# B&R Automation Studio project BenchEDM_AS6 (part 8)

#### OMD_MR.st
```iecst
ACTION OMD_MR:

	FOR i := 0 TO MAX_DRIVER_MR_IDX DO
		IF NOT gDriver.MR[i].FirstScanComplete THEN
			gDriver.MR[i].FirstScanComplete 			:= TRUE;
			gDriver.MR[i].DefaultPar.Device				:= 'SL2.IF1.ST1.IF1.ST5.IF1';					//ST
			gDriver.MR[i].DefaultPar.Mode				:= '/PHY=RS485 /PA=E /DB=8 /SB=1 /BD=38400';	//ST
			gDriver.MR[i].DefaultPar.DataObject			:= 'MbRTU';										//ST
			gDriver.MR[i].DefaultPar.IsAscii			:= FALSE;										//BO
			gDriver.MR[i].DefaultPar.Timeout			:= 1.0;											//LR
			gDriver.MR[i].DefaultPar.CmdNode			:= 1;											//UD
			gDriver.MR[i].DefaultPar.CmdFunctionCall	:= 1;											//UD
			gDriver.MR[i].DefaultPar.CmdOffset			:= 1;											//UD
			gDriver.MR[i].DefaultPar.CmdData			:= 0;											//UD
			brsmemcpy(ADR(gDriver.MR[i].Par),ADR(gDriver.MR[i].DefaultPar),SIZEOF(gDriver.MR[i].Par));
		ELSIF NOT gDriver.MR[i].ParametersLoaded AND gMain.Services.Recipes.Out.ParametersReady THEN
			gDriver.MR[i].ParametersLoaded := TRUE;
			brsmemcpy(ADR(gDriver.MR[i].Par),ADR(gPar.Driver.MR[i]),SIZEOF(gDriver.MR[i].Par));
		END_IF;

		brsmemset(ADR(gDriver.MR[i].Sev),0,SIZEOF(gDriver.MR[i].Sev));
		brsmemset(ADR(gDriver.MR[i].Status),0,SIZEOF(gDriver.MR[i].Status));
		FOR j := 0 TO MAX_DRIVER_MR_MON_IDX DO
			IF gDriver.MR[i].Par.Mon[j].Enable THEN
				IF gDriver.MR[i].Mon[j] THEN
					gDriver.MR[i].CTON_Mon[j](IN := TRUE, PT := LREAL_TO_TIME(gDriver.MR[i].Par.Mon[j].Time*1000.0));
					IF gDriver.MR[i].CTON_Mon[j].Q THEN
						gDriver.MR[i].Sev[j] := gDriver.MR[i].Par.Mon[j].Sev;
						IF gDriver.MR[i].Status.Severity < gDriver.MR[i].Sev[j] THEN
							gDriver.MR[i].Status.Severity := gDriver.MR[i].Sev[j];
						END_IF;
					END_IF;
				ELSE
					gDriver.MR[i].CTON_Mon[j](IN := FALSE);
					gDriver.MR[i].Sev[j] := 0;
				END_IF;
			ELSE
				gDriver.MR[i].CTON_Mon[j](IN := FALSE);
				gDriver.MR[i].Sev[j] := 0;
			END_IF;
		END_FOR;
		IF gDriver.MR[i].Cmd[C_MR_RESET] OR gDriver.ResetAll THEN
			gDriver.MR[i].Cmd[C_MR_RESET] := FALSE;
			brsmemset(ADR(gDriver.MR[i].Mon),0,SIZEOF(gDriver.MR[i].Mon));
			brsmemset(ADR(gDriver.MR[i].Cmd),0,SIZEOF(gDriver.MR[i].Cmd));
			brsmemset(ADR(gDriver.MR[i].Sev),0,SIZEOF(gDriver.MR[i].Sev));
			brsmemset(ADR(gDriver.MR[i].Status),0,SIZEOF(gDriver.MR[i].Status));
		END_IF;
		IF gDriver.MR[i].Cmd[C_MR_CLEARCMD] THEN
			gDriver.MR[i].Cmd[C_MR_CLEARCMD] := FALSE;
			brsmemset(ADR(gDriver.MR[i].Cmd),0,SIZEOF(gDriver.MR[i].Cmd));
		END_IF;
		IF gDriver.MR[i].Cmd[C_MR_CLEARMON] THEN
			gDriver.MR[i].Cmd[C_MR_CLEARMON] := FALSE;
			brsmemset(ADR(gDriver.MR[i].Status.Severity),0,SIZEOF(gDriver.MR[i].Status.Severity));
			brsmemset(ADR(gDriver.MR[i].Sev),0,SIZEOF(gDriver.MR[i].Sev));
			brsmemset(ADR(gDriver.MR[i].Par.Mon),0,SIZEOF(gDriver.MR[i].Par.Mon));
		END_IF;
		IF gDriver.MR[i].Cmd[C_MR_DEFAULTMON] THEN
			gDriver.MR[i].Cmd[C_MR_DEFAULTMON] := FALSE;
			brsmemcpy(ADR(gDriver.MR[i].Par.Mon),ADR(gDriver.MR[i].DefaultPar.Mon),SIZEOF(gDriver.MR[i].Par.Mon));
		END_IF;
		IF gDriver.MR[i].Cmd[C_MR_CLEARPAR] THEN
			gDriver.MR[i].Cmd[C_MR_CLEARPAR] := FALSE;
			brsmemset(ADR(gDriver.MR[i].Par),0,SIZEOF(gDriver.MR[i].Par));
		END_IF;
		IF gDriver.MR[i].Cmd[C_MR_DEFAULTPAR] THEN
			gDriver.MR[i].Cmd[C_MR_DEFAULTPAR] := FALSE;
			brsmemcpy(ADR(gDriver.MR[i].Par),ADR(gDriver.MR[i].DefaultPar),SIZEOF(gDriver.MR[i].Par));
		END_IF;
		IF gDriver.MR[i].Cmd[C_MR_SAVEPAR] THEN
			gDriver.MR[i].Cmd[C_MR_SAVEPAR] := FALSE;
			brsmemcpy(ADR(gPar.Driver.MR[i]),ADR(gDriver.MR[i].Par),SIZEOF(gDriver.MR[i].Par));
		END_IF;
		IF gDriver.MR[i].Cmd[C_MR_LOADPAR] THEN
			gDriver.MR[i].Cmd[C_MR_LOADPAR] := FALSE;
			brsmemcpy(ADR(gDriver.MR[i].Par),ADR(gPar.Driver.MR[i]),SIZEOF(gDriver.MR[i].Par));
		END_IF;

		gDriver.MR[i].MBMOpen_0.enable					:= gDriver.MR[i].Cmd[C_MR_MBMOPEN] AND NOT (gDriver.MR[i].Cmd[C_MR_ERRORRESET] OR gMain.ErrorReset);
		gDriver.MR[i].MBMaster_0.enable					:= gDriver.MR[i].Cmd[C_MR_MBMASTER] AND NOT (gDriver.MR[i].Cmd[C_MR_ERRORRESET] OR gMain.ErrorReset);
		gDriver.MR[i].MBMCmd_0.enable					:= gDriver.MR[i].Cmd[C_MR_MBMCMD] AND NOT (gDriver.MR[i].Cmd[C_MR_ERRORRESET] OR gMain.ErrorReset);
		gDriver.MR[i].MBMClose_0.enable					:= gDriver.MR[i].Cmd[C_MR_MBMCLOSE] AND NOT (gDriver.MR[i].Cmd[C_MR_ERRORRESET] OR gMain.ErrorReset);

		gDriver.MR[i].MBMOpen_0(pDevice := ADR(gDriver.MR[i].Par.Device), pMode := ADR(gDriver.MR[i].Par.Mode), pConfig := ADR(gDriver.MR[i].Par.DataObject), timeout := LREAL_TO_UINT(gDriver.MR[i].Par.Timeout*1000.0), ascii := BOOL_TO_USINT(gDriver.MR[i].Par.IsAscii));
		IF gDriver.MR[i].MBMOpen_0.ident <> 0 AND gDriver.MR[i].MBMOpen_0.enable THEN
			gDriver.MR[i].Ident := gDriver.MR[i].MBMOpen_0.ident;
		END_IF;
		gDriver.MR[i].MBMCmd_0(ident := gDriver.MR[i].Ident, mfc := UDINT_TO_USINT(gDriver.MR[i].Par.CmdFunctionCall), node := UDINT_TO_USINT(gDriver.MR[i].Par.CmdNode), data := ADR(gDriver.MR[i].Par.CmdData), offset := UDINT_TO_UINT(gDriver.MR[i].Par.CmdOffset), len := 1);
		gDriver.MR[i].MBMaster_0(ident := gDriver.MR[i].Ident);
		gDriver.MR[i].MBMClose_0(ident := gDriver.MR[i].Ident);
		IF gDriver.MR[i].MBMClose_0.enable AND gDriver.MR[i].MBMClose_0.status = 0 THEN
			gDriver.MR[i].Ident := 0;
		END_IF;

		gDriver.MR[i].Status.Active						:= gDriver.MR[i].MBMaster_0.enable AND (gDriver.MR[i].MBMaster_0.status = 65535 OR gDriver.MR[i].MBMaster_0.status = 0);

		gDriver.MR[i].Wait[W_MR_NOERROR]				:= BOOL_TO_DINT((gDriver.MR[i].MBMOpen_0.status = 0 OR gDriver.MR[i].MBMOpen_0.status = 65535 OR gDriver.MR[i].MBMOpen_0.status = 65534) AND (gDriver.MR[i].MBMaster_0.status = 0 OR gDriver.MR[i].MBMaster_0.status = 65535 OR gDriver.MR[i].MBMaster_0.status = 65534) AND (gDriver.MR[i].MBMCmd_0.status = 0 OR gDriver.MR[i].MBMCmd_0.status = 65535 OR gDriver.MR[i].MBMCmd_0.status = 65534) AND (gDriver.MR[i].MBMClose_0.status = 0 OR gDriver.MR[i].MBMClose_0.status = 65535 OR gDriver.MR[i].MBMClose_0.status = 65534));
		gDriver.MR[i].Wait[W_MR_MBMOPEN]				:= BOOL_TO_DINT(gDriver.MR[i].MBMOpen_0.status = 0);
		gDriver.MR[i].Wait[W_MR_MBMASTER]				:= BOOL_TO_DINT(gDriver.MR[i].MBMaster_0.status = 0 OR gDriver.MR[i].MBMaster_0.status = 65535);
		gDriver.MR[i].Wait[W_MR_MBMCMD]					:= BOOL_TO_DINT(gDriver.MR[i].MBMCmd_0.status = 0);
		gDriver.MR[i].Wait[W_MR_MBMCLOSE]				:= BOOL_TO_DINT(gDriver.MR[i].MBMClose_0.status = 0);

		IF gDriver.MR[i].MBMaster_0.enable THEN
			IF gDriver.MR[i].Wait[W_MR_NOERROR] = 0 THEN
				gDriver.MR[i].Mon[M_MR_ERROR]			:= TRUE;
			ELSIF gDriver.MR[i].MBMaster_0.execute THEN
				gDriver.MR[i].Mon[M_MR_ERROR]			:= FALSE;
			END_IF;
		ELSE
			gDriver.MR[i].Mon[M_MR_ERROR]				:= gDriver.MR[i].Wait[W_MR_NOERROR] = 0;
		END_IF;
	END_FOR;

END_ACTION
```

#### OMD_BX.st
```iecst
ACTION OMD_BX:

	FOR i := 0 TO MAX_DRIVER_BX_IDX DO
		IF NOT gDriver.BX[i].FirstScanComplete THEN
			gDriver.BX[i].FirstScanComplete 				:= TRUE;
			gDriver.BX[i].DefaultPar.EdgeFindMode			:= FALSE; 	//BO
			gDriver.BX[i].DefaultPar.ISOPulseMode			:= FALSE; 	//BO
			gDriver.BX[i].DefaultPar.ElectrodePositiveMode	:= FALSE; 	//BO
			gDriver.BX[i].DefaultPar.Current				:= 15.0; 	//RR
			gDriver.BX[i].DefaultPar.OnTime					:= 3.0; 	//RR
			gDriver.BX[i].DefaultPar.OffTime				:= 27.0; 	//RR
			gDriver.BX[i].DefaultPar.SetFeedback			:= 75.0; 	//RR
			gDriver.BX[i].DefaultPar.MinOverrideFactor		:= -200.0; 	//RR
			gDriver.BX[i].DefaultPar.MaxOverrideFactor		:= 200.0; 	//RR
			gDriver.BX[i].DefaultPar.PID.Gain				:= 0.1; 	//RR
			gDriver.BX[i].DefaultPar.PID.IntegrationTime	:= 0.0; 	//RR
			gDriver.BX[i].DefaultPar.PID.DerivativeTime		:= 0.0; 	//RR
			gDriver.BX[i].DefaultPar.PID.FilterTime			:= 0.0; 	//RR
			brsmemcpy(ADR(gDriver.BX[i].Par),ADR(gDriver.BX[i].DefaultPar),SIZEOF(gDriver.BX[i].Par));
		ELSIF NOT gDriver.BX[i].ParametersLoaded AND gMain.Services.Recipes.Out.ParametersReady THEN
			gDriver.BX[i].ParametersLoaded 					:= TRUE;
			brsmemcpy(ADR(gDriver.BX[i].Par),ADR(gPar.Driver.BX[i]),SIZEOF(gDriver.BX[i].Par));
		END_IF;

		brsmemset(ADR(gDriver.BX[i].Sev),0,SIZEOF(gDriver.BX[i].Sev));
		brsmemset(ADR(gDriver.BX[i].Status),0,SIZEOF(gDriver.BX[i].Status));
		FOR j := 0 TO MAX_DRIVER_BX_MON_IDX DO
			IF gDriver.BX[i].Par.Mon[j].Enable THEN
				IF gDriver.BX[i].Mon[j] THEN
					gDriver.BX[i].CTON_Mon[j](IN := TRUE, PT := LREAL_TO_TIME(gDriver.BX[i].Par.Mon[j].Time*1000.0));
					IF gDriver.BX[i].CTON_Mon[j].Q THEN
						gDriver.BX[i].Sev[j] 				:= gDriver.BX[i].Par.Mon[j].Sev;
						IF gDriver.BX[i].Status.Severity < gDriver.BX[i].Sev[j] THEN
							gDriver.BX[i].Status.Severity 	:= gDriver.BX[i].Sev[j];
						END_IF;
					END_IF;
				ELSE
					gDriver.BX[i].CTON_Mon[j](IN := FALSE);
					gDriver.BX[i].Sev[j] 					:= 0;
				END_IF;
			ELSE
				gDriver.BX[i].CTON_Mon[j](IN := FALSE);
				gDriver.BX[i].Sev[j] 						:= 0;
			END_IF;
		END_FOR;
		IF gDriver.BX[i].Cmd[C_BX_RESET] OR gDriver.ResetAll THEN
			gDriver.BX[i].Cmd[C_BX_RESET] 					:= FALSE;
			brsmemset(ADR(gDriver.BX[i].Mon),0,SIZEOF(gDriver.BX[i].Mon));
			brsmemset(ADR(gDriver.BX[i].Cmd),0,SIZEOF(gDriver.BX[i].Cmd));
			brsmemset(ADR(gDriver.BX[i].Sev),0,SIZEOF(gDriver.BX[i].Sev));
			brsmemset(ADR(gDriver.BX[i].Status),0,SIZEOF(gDriver.BX[i].Status));
		END_IF;
		IF gDriver.BX[i].Cmd[C_BX_CLEARCMD] THEN
			gDriver.BX[i].Cmd[C_BX_CLEARCMD] 				:= FALSE;
			brsmemset(ADR(gDriver.BX[i].Cmd),0,SIZEOF(gDriver.BX[i].Cmd));
		END_IF;
		IF gDriver.BX[i].Cmd[C_BX_CLEARMON] THEN
			gDriver.BX[i].Cmd[C_BX_CLEARMON] 				:= FALSE;
			brsmemset(ADR(gDriver.BX[i].Status.Severity),0,SIZEOF(gDriver.BX[i].Status.Severity));
			brsmemset(ADR(gDriver.BX[i].Sev),0,SIZEOF(gDriver.BX[i].Sev));
			brsmemset(ADR(gDriver.BX[i].Par.Mon),0,SIZEOF(gDriver.BX[i].Par.Mon));
		END_IF;
		IF gDriver.BX[i].Cmd[C_BX_DEFAULTMON] THEN
			gDriver.BX[i].Cmd[C_BX_DEFAULTMON] 				:= FALSE;
			brsmemcpy(ADR(gDriver.BX[i].Par.Mon),ADR(gDriver.BX[i].DefaultPar.Mon),SIZEOF(gDriver.BX[i].Par.Mon));
		END_IF;
		IF gDriver.BX[i].Cmd[C_BX_CLEARPAR] THEN
			gDriver.BX[i].Cmd[C_BX_CLEARPAR] 				:= FALSE;
			brsmemset(ADR(gDriver.BX[i].Par),0,SIZEOF(gDriver.BX[i].Par));
		END_IF;
		IF gDriver.BX[i].Cmd[C_BX_DEFAULTPAR] THEN
			gDriver.BX[i].Cmd[C_BX_DEFAULTPAR] 				:= FALSE;
			brsmemcpy(ADR(gDriver.BX[i].Par),ADR(gDriver.BX[i].DefaultPar),SIZEOF(gDriver.BX[i].Par));
		END_IF;
		IF gDriver.BX[i].Cmd[C_BX_SAVEPAR] THEN
			gDriver.BX[i].Cmd[C_BX_SAVEPAR] 				:= FALSE;
			brsmemcpy(ADR(gPar.Driver.BX[i]),ADR(gDriver.BX[i].Par),SIZEOF(gDriver.BX[i].Par));
		END_IF;
		IF gDriver.BX[i].Cmd[C_BX_LOADPAR] THEN
			gDriver.BX[i].Cmd[C_BX_LOADPAR] 				:= FALSE;
			brsmemcpy(ADR(gDriver.BX[i].Par),ADR(gPar.Driver.BX[i]),SIZEOF(gDriver.BX[i].Par));
		END_IF;

		gDriver.BX[i].Status.SetOffTime						:= gDriver.BX[i].Par.OffTime;
		gDriver.BX[i].Status.SetOnTime						:= gDriver.BX[i].Par.OnTime;
		gDriver.BX[i].Status.SetCurrent						:= gDriver.BX[i].Par.Current;
		gDriver.BX[i].Status.SetFeedback					:= gDriver.BX[i].Par.SetFeedback;
		gDriver.BX[i].Status.ActualPower					:= LREAL_TO_REAL(gIO.BX18.TC_IO_AI_Power.Signal.Filtered);
		gDriver.BX[i].Status.ActualFeedback					:= LREAL_TO_REAL(gIO.BX18.TC_IO_AI_Feedback.Signal.Filtered);
		gDriver.BX[i].Status.OutputActive					:= gIO.BX18.TC_IO_DI_EDMOutputActive.Signal.Filtered;
		gDriver.BX[i].Status.EdgeFindEnabled				:= gIO.BX18.TC_IO_DI_EdgefindModeEnabled.Signal.Filtered;
		gDriver.BX[i].Status.EdgeFound						:= gIO.BX18.TC_IO_DI_EdgeFound.Signal.Filtered;
		gDriver.BX[i].Status.StateInvalid					:= gIO.BX18.TC_IO_DI_ReqStateInvalid.Signal.Filtered;
		gDriver.BX[i].Status.SettingsInvalid				:= gIO.BX18.TC_IO_DI_ReqSettingsInvalid.Signal.Filtered;
		gDriver.BX[i].Status.PowerFault						:= gIO.BX18.TC_IO_DI_PowerFault.Signal.Filtered;
		gDriver.BX[i].Status.LowVoltageFault				:= gIO.BX18.TC_IO_DI_LowVoltageFault.Signal.Filtered;
		gDriver.BX[i].Status.HighVoltageFault				:= gIO.BX18.TC_IO_DI_HighVoltageFault.Signal.Filtered;
		gDriver.BX[i].Status.EstopActive					:= gIO.BX18.TC_IO_DI_EstopActive.Signal.Filtered;
		gDriver.BX[i].Status.ISOPulseMode					:= gIO.BX18.TC_IO_DI_ISOPulseMode.Signal.Filtered;
		gDriver.BX[i].Status.ElectrodePositiveMode			:= gIO.BX18.TC_IO_DI_ElectrodePositiveMode.Signal.Filtered;

		IF gDriver.BX[i].MTBasicsPID_0.PIDParameters.Gain <> gDriver.BX[i].Par.PID.Gain OR gDriver.BX[i].MTBasicsPID_0.PIDParameters.IntegrationTime <> gDriver.BX[i].Par.PID.IntegrationTime OR gDriver.BX[i].MTBasicsPID_0.PIDParameters.DerivativeTime <> gDriver.BX[i].Par.PID.DerivativeTime OR gDriver.BX[i].MTBasicsPID_0.PIDParameters.FilterTime <> gDriver.BX[i].Par.PID.FilterTime OR gDriver.BX[i].MTBasicsPID_0.MinOut <> gDriver.BX[i].Par.MinOverrideFactor OR gDriver.BX[i].MTBasicsPID_0.MaxOut <> gDriver.BX[i].Par.MaxOverrideFactor THEN
			gDriver.BX[i].MTBasicsPID_0.Update 				:= TRUE;
		END_IF;
		gDriver.BX[i].MTBasicsPID_0(Enable := gDriver.BX[i].Cmd[C_BX_ENABLE] AND gDriver.BX[i].Wait[W_BX_NOERROR] = 1, PIDParameters := gDriver.BX[i].Par.PID, MinOut := gDriver.BX[i].Par.MinOverrideFactor, MaxOut := gDriver.BX[i].Par.MaxOverrideFactor, SetValue := gDriver.BX[i].Par.SetFeedback, ActValue := gDriver.BX[i].Status.ActualFeedback, Invert := TRUE);
		gDriver.BX[i].MTBasicsPID_0.Update 					:= FALSE;

		gDriver.BX[i].Status.OverrideFactor					:= gDriver.BX[i].MTBasicsPID_0.Out;

		gDriver.BX[i].Wait[W_BX_NOERROR]					:= BOOL_TO_DINT(NOT gDriver.BX[i].Status.StateInvalid AND NOT gDriver.BX[i].Status.SettingsInvalid AND NOT gDriver.BX[i].Status.PowerFault AND NOT gDriver.BX[i].Status.LowVoltageFault AND NOT gDriver.BX[i].Status.HighVoltageFault AND NOT gDriver.BX[i].Status.EstopActive);
		gDriver.BX[i].Wait[W_BX_ACTIVE]						:= BOOL_TO_DINT(gDriver.BX[i].Wait[W_BX_NOERROR] = 1 AND gDriver.BX[i].Status.OutputActive);
		gDriver.BX[i].Mon[M_BX_ERROR]						:= gDriver.BX[i].Wait[W_BX_NOERROR] <> 1;

		gIO.BX18.TC_IO_AO_Current.Logical					:= gDriver.BX[i].Par.Current;
		gIO.BX18.TC_IO_AO_OffTime.Logical					:= gDriver.BX[i].Par.OffTime;
		gIO.BX18.TC_IO_AO_OnTime.Logical					:= gDriver.BX[i].Par.OnTime;
		gIO.BX18.TC_IO_DO_ChangeRequest.Logical				:= gIO.BX18.TC_IO_DI_CurrentChanged.Signal.Filtered OR gIO.BX18.TC_IO_DI_OnTimeChanged.Signal.Filtered OR gIO.BX18.TC_IO_DI_OffTimeChanged.Signal.Filtered;
		gIO.BX18.TC_IO_DO_EdgeFindMode.Logical				:= gDriver.BX[i].Par.EdgeFindMode;
		gIO.BX18.TC_IO_DO_ElectrodePositiveMode.Logical		:= gDriver.BX[i].Par.ElectrodePositiveMode;
		gIO.BX18.TC_IO_DO_ISOFreqMode.Logical				:= gDriver.BX[i].Par.ISOPulseMode;
		gIO.BX18.TC_IO_DO_Enable.Logical					:= gDriver.BX[i].Cmd[C_BX_ENABLE];
	END_FOR;

END_ACTION
```

#### OMD_IO.st - not listed in the package file held
```iecst
ACTION OMD_IO:

	FOR i := 0 TO MAX_DRIVER_AB_IDX DO
		IF NOT gDriver.AB[i].FirstScanComplete THEN
			gDriver.AB[i].FirstScanComplete 													:= TRUE;
			gDriver.AB[i].DefaultPar.AB.Acceleration											:= 50.0;							//RR
			gDriver.AB[i].DefaultPar.AB.AutoTune.FeedForward.Acceleration						:= 50.0;							//RR
			gDriver.AB[i].DefaultPar.AB.AutoTune.FeedForward.Direction							:= mcDIR_BOTH;						//McDirectionEnum
			gDriver.AB[i].DefaultPar.AB.AutoTune.FeedForward.MaxVelocityPercent					:= 50.0;							//RR
			gDriver.AB[i].DefaultPar.AB.AutoTune.FeedForward.Mode								:= mcACPAX_TUNE_FF_MODE_STANDARD; 	//McAcpAxAutoTuneFeedFwdModeEnum
			gDriver.AB[i].DefaultPar.AB.AutoTune.LoopFilterMode									:= mcAXIS_TUNE_LOOP_FILTER_F1;		//MpAxisAutoTuneLoopFilterModeEnum
			gDriver.AB[i].DefaultPar.AB.AutoTune.MaxCurrentPercent								:= 80.0;							//RR
			gDriver.AB[i].DefaultPar.AB.AutoTune.MaxDistance									:= 0.0;								//LR
			gDriver.AB[i].DefaultPar.AB.AutoTune.MaxPositionError								:= 1.0;								//LR
			gDriver.AB[i].DefaultPar.AB.AutoTune.Mode											:= mcAXIS_TUNE_AUTOMATIC;			//MpAxisAutoTuneModeEnum
			gDriver.AB[i].DefaultPar.AB.AutoTune.Options.MaxProportionalGain					:= 0.0;								//RR
			gDriver.AB[i].DefaultPar.AB.AutoTune.Options.SpeedTuneFilterTmeMode					:= mcACPAX_FILTER_TIME_USE;			//McAcpAxFilterTimeModeEnum
			gDriver.AB[i].DefaultPar.AB.AutoTune.Options.SpeedTuneLoopFilter1Mode				:= mcACPAX_LOOP_FILTER_IGNORE;		//McAcpAxLoopFilterModeEnum
			gDriver.AB[i].DefaultPar.AB.AutoTune.Orientation									:= mcACPAX_ORIENTATION_HORIZONTAL;	//McAcpAxAutoTuneOrientationEnum
			gDriver.AB[i].DefaultPar.AB.AutoTune.SaveControllerSettings							:= FALSE;							//BO
			gDriver.AB[i].DefaultPar.AB.Deceleration											:= 50.0;							//RR
			gDriver.AB[i].DefaultPar.AB.Direction												:= mcDIR_SHORTEST_WAY;				//McDirectionEnum
			gDriver.AB[i].DefaultPar.AB.Distance												:= 0.0;								//LR
			gDriver.AB[i].DefaultPar.AB.Homing.Mode												:= mcHOMING_DIRECT;					//McHomingModeEnum
			gDriver.AB[i].DefaultPar.AB.Homing.Position											:= 0.0;								//RR
			gDriver.AB[i].DefaultPar.AB.Homing.Options.Acceleration								:= 50.0;							//RR
			gDriver.AB[i].DefaultPar.AB.Homing.Options.AdditionalTorqueLimit.NegativeDirection	:= 0.0;								//RR
			gDriver.AB[i].DefaultPar.AB.Homing.Options.AdditionalTorqueLimit.PositiveDirection	:= 0.0;								//RR
			gDriver.AB[i].DefaultPar.AB.Homing.Options.BlockDetectionPositionError				:= 0.0;								//RR
			gDriver.AB[i].DefaultPar.AB.Homing.Options.DisableRestorePositionOnEnable			:= mcSWITCH_OFF;					//McSwitchEnum
			gDriver.AB[i].DefaultPar.AB.Homing.Options.DriveSpecificHoming						:= mcSWITCH_OFF;					//McSwitchEnum
			gDriver.AB[i].DefaultPar.AB.Homing.Options.DriveSpecificHomingMode					:= 0;								//SS
			gDriver.AB[i].DefaultPar.AB.Homing.Options.HomingDirection							:= mcDIR_POSITIVE;					//McDirectionEnum
			gDriver.AB[i].DefaultPar.AB.Homing.Options.HomingVelocity							:= 5.0;								//RR
			gDriver.AB[i].DefaultPar.AB.Homing.Options.KeepDirection							:= mcSWITCH_OFF;					//McSwitchEnum
			gDriver.AB[i].DefaultPar.AB.Homing.Options.PositionErrorStopLimit					:= 0.0;								//RR
			gDriver.AB[i].DefaultPar.AB.Homing.Options.ReferencePulse							:= mcSWITCH_OFF;					//McSwitchEnum
			gDriver.AB[i].DefaultPar.AB.Homing.Options.ReferencePulseBlockingDistance			:= 0.0;								//RR
			gDriver.AB[i].DefaultPar.AB.Homing.Options.RestorePositionVariableAddress			:= 0;								//UD
			gDriver.AB[i].DefaultPar.AB.Homing.Options.SensorOffset								:= 0.0;								//LR
			gDriver.AB[i].DefaultPar.AB.Homing.Options.SensorOffsetDirection					:= mcDIR_POSITIVE;					//McDirectionEnum
			gDriver.AB[i].DefaultPar.AB.Homing.Options.StartDirection							:= mcDIR_POSITIVE;					//McDirectionEnum
			gDriver.AB[i].DefaultPar.AB.Homing.Options.StartVelocity							:= 1.0;								//RR
			gDriver.AB[i].DefaultPar.AB.Homing.Options.SwitchEdge								:= mcDIR_POSITIVE;					//McDirectionEnum
			gDriver.AB[i].DefaultPar.AB.Homing.Options.TorqueLimit								:= 0.1;								//RR
			gDriver.AB[i].DefaultPar.AB.Jerk													:= 0.0;								//RR
			gDriver.AB[i].DefaultPar.AB.Jog.Acceleration										:= 50.0;							//RR
			gDriver.AB[i].DefaultPar.AB.Jog.Deceleration										:= 50.0;							//RR
			gDriver.AB[i].DefaultPar.AB.Jog.Jerk												:= 0.0;								//RR
			gDriver.AB[i].DefaultPar.AB.Jog.LimitPosition.FirstPosition							:= 0.0;								//LR
			gDriver.AB[i].DefaultPar.AB.Jog.LimitPosition.LastPosition							:= 0.0;								//LR
			gDriver.AB[i].DefaultPar.AB.Jog.Velocity											:= 5.0;								//RR
			gDriver.AB[i].DefaultPar.AB.LimitLoad.Direction										:= mcDIR_CURRENT;					//McDirectionEnum
			gDriver.AB[i].DefaultPar.AB.LimitLoad.Load											:= 2.0;								//RR
			gDriver.AB[i].DefaultPar.AB.Position												:= 0.0;								//LR
			gDriver.AB[i].DefaultPar.AB.Stop.Deceleration										:= 50.0;							//RR
			gDriver.AB[i].DefaultPar.AB.Stop.Jerk												:= 0.0;								//RR
			gDriver.AB[i].DefaultPar.AB.Stop.StopAtPosition.Activate							:= FALSE;							//BO
			gDriver.AB[i].DefaultPar.AB.Stop.StopAtPosition.Deceleration						:= 0.0;								//RR
			gDriver.AB[i].DefaultPar.AB.Stop.StopAtPosition.Position							:= 0.0;								//LR
			gDriver.AB[i].DefaultPar.AB.Velocity												:= 5.0;								//RR

			brsmemcpy(ADR(gDriver.AB[i].Par),ADR(gDriver.AB[i].DefaultPar),SIZEOF(gDriver.AB[i].Par));
		END_IF;

		brsmemset(ADR(gDriver.AB[i].Sev),0,SIZEOF(gDriver.AB[i].Sev));
		brsmemset(ADR(gDriver.AB[i].Status),0,SIZEOF(gDriver.AB[i].Status));
		FOR j := 0 TO MAX_DRIVER_AB_MON_IDX DO
			IF gDriver.AB[i].Par.Mon[j].Enable THEN
				IF gDriver.AB[i].Mon[j] THEN
					gDriver.AB[i].CTON_Mon[j](IN := TRUE, PT := LREAL_TO_TIME(gDriver.AB[i].Par.Mon[j].Time*1000.0));
					IF gDriver.AB[i].CTON_Mon[j].Q THEN
						gDriver.AB[i].Sev[j] := gDriver.AB[i].Par.Mon[j].Sev;
						IF gDriver.AB[i].Status.Severity < gDriver.AB[i].Sev[j] THEN
							gDriver.AB[i].Status.Severity := gDriver.AB[i].Sev[j];
						END_IF;
					END_IF;
				ELSE
					gDriver.AB[i].CTON_Mon[j](IN := FALSE);
					gDriver.AB[i].Sev[j] := 0;
				END_IF;
			ELSE
				gDriver.AB[i].CTON_Mon[j](IN := FALSE);
				gDriver.AB[i].Sev[j] := 0;
			END_IF;
		END_FOR;
		IF gDriver.AB[i].Cmd[C_AB_RESET] THEN
			gDriver.AB[i].Cmd[C_AB_RESET] := FALSE;
			brsmemset(ADR(gDriver.AB[i].Cmd),0,SIZEOF(gDriver.AB[i].Cmd));
			brsmemset(ADR(gDriver.AB[i].Sev),0,SIZEOF(gDriver.AB[i].Sev));
			brsmemset(ADR(gDriver.AB[i].Status),0,SIZEOF(gDriver.AB[i].Status));
			brsmemcpy(ADR(gDriver.AB[i].Par),ADR(gDriver.AB[i].DefaultPar),SIZEOF(gDriver.AB[i].Par));
		END_IF;
		IF gDriver.AB[i].Cmd[C_AB_CLEARCMD] THEN
			gDriver.AB[i].Cmd[C_AB_CLEARCMD] := FALSE;
			brsmemset(ADR(gDriver.AB[i].Cmd),0,SIZEOF(gDriver.AB[i].Cmd));
		END_IF;
		IF gDriver.AB[i].Cmd[C_AB_CLEARMON] THEN
			gDriver.AB[i].Cmd[C_AB_CLEARMON] := FALSE;
			brsmemset(ADR(gDriver.AB[i].Status.Severity),0,SIZEOF(gDriver.AB[i].Status.Severity));
			brsmemset(ADR(gDriver.AB[i].Sev),0,SIZEOF(gDriver.AB[i].Sev));
			brsmemset(ADR(gDriver.AB[i].Par.Mon),0,SIZEOF(gDriver.AB[i].Par.Mon));
		END_IF;
		IF gDriver.AB[i].Cmd[C_AB_DEFAULTMON] THEN
			gDriver.AB[i].Cmd[C_AB_DEFAULTMON] := FALSE;
			brsmemcpy(ADR(gDriver.AB[i].Par.Mon),ADR(gDriver.AB[i].DefaultPar.Mon),SIZEOF(gDriver.AB[i].Par.Mon));
		END_IF;
		IF gDriver.AB[i].Cmd[C_AB_CLEARPAR] THEN
			gDriver.AB[i].Cmd[C_AB_CLEARPAR] := FALSE;
			brsmemset(ADR(gDriver.AB[i].Par),0,SIZEOF(gDriver.AB[i].Par));
		END_IF;
		IF gDriver.AB[i].Cmd[C_AB_DEFAULTPAR] THEN
			gDriver.AB[i].Cmd[C_AB_DEFAULTPAR] := FALSE;
			brsmemcpy(ADR(gDriver.AB[i].Par),ADR(gDriver.AB[i].DefaultPar),SIZEOF(gDriver.AB[i].Par));
		END_IF;
		gDriver.AB[i].MpAxisBasic_0.ErrorReset			:= gDriver.AB[i].Cmd[C_AB_ERRORRESET] OR gMain.ErrorReset;
		gDriver.AB[i].MpAxisBasic_0.Home				:= gDriver.AB[i].Cmd[C_AB_HOME];
		gDriver.AB[i].MpAxisBasic_0.Power				:= gDriver.AB[i].Cmd[C_AB_POWER];
		gDriver.AB[i].MpAxisBasic_0.Update				:= gDriver.AB[i].Cmd[C_AB_UPDATE];
		gDriver.AB[i].MpAxisBasic_0.AutoTune			:= gDriver.AB[i].Cmd[C_AB_AUTOTUNE];
		gDriver.AB[i].MpAxisBasic_0.JogPositive			:= gDriver.AB[i].Cmd[C_AB_JOGPOSITIVE];
		gDriver.AB[i].MpAxisBasic_0.JogNegative			:= gDriver.AB[i].Cmd[C_AB_JOGNEGATIVE];
		gDriver.AB[i].MpAxisBasic_0.LimitLoad			:= gDriver.AB[i].Cmd[C_AB_LIMITLOAD];
		gDriver.AB[i].MpAxisBasic_0.Stop				:= gDriver.AB[i].Cmd[C_AB_STOP];
		gDriver.AB[i].MpAxisBasic_0.MoveAbsolute		:= gDriver.AB[i].Cmd[C_AB_MOVEABSOLUTE];
		gDriver.AB[i].MpAxisBasic_0.MoveAdditive		:= gDriver.AB[i].Cmd[C_AB_MOVEADDITIVE];
		gDriver.AB[i].MpAxisBasic_0.MoveVelocity		:= gDriver.AB[i].Cmd[C_AB_MOVEVELOCITY];
		gDriver.AB[i].MpAxisBasic_0.ReleaseBrake		:= gDriver.AB[i].Cmd[C_AB_RELEASEBRAKE];
		gDriver.AB[i].MpAxisBasic_0.Simulate			:= gDriver.AB[i].Cmd[C_AB_SIMULATE];

		gDriver.AB[i].MpAxisBasic_0(MpLink := gDriver.AB[i].MpLinkADR, Enable := TRUE, Parameters := ADR(gDriver.AB[i].Par.AB));

		gDriver.AB[i].Status.Position					:= gDriver.AB[i].MpAxisBasic_0.Position;
		gDriver.AB[i].Status.Velocity					:= gDriver.AB[i].MpAxisBasic_0.Velocity;

		gDriver.AB[i].Wait[W_AB_NOERROR]				:= BOOL_TO_DINT(NOT gDriver.AB[i].MpAxisBasic_0.Error);
		gDriver.AB[i].Wait[W_AB_COMMUNICATIONREADY]		:= BOOL_TO_DINT(gDriver.AB[i].MpAxisBasic_0.Info.CommunicationReady);
		gDriver.AB[i].Wait[W_AB_READYTOPOWERON]			:= BOOL_TO_DINT(gDriver.AB[i].MpAxisBasic_0.Info.ReadyToPowerOn);
		gDriver.AB[i].Wait[W_AB_POWERON]				:= BOOL_TO_DINT(gDriver.AB[i].MpAxisBasic_0.PowerOn);
		gDriver.AB[i].Wait[W_AB_ISHOMED]				:= BOOL_TO_DINT(gDriver.AB[i].MpAxisBasic_0.IsHomed AND NOT gDriver.AB[i].MpAxisBasic_0.CommandBusy);
		gDriver.AB[i].Wait[W_AB_LIMITLOADACTIVE]		:= BOOL_TO_DINT(gDriver.AB[i].MpAxisBasic_0.LimitLoadReady);
		gDriver.AB[i].Wait[W_AB_MOVEDONE]				:= BOOL_TO_DINT(gDriver.AB[i].MpAxisBasic_0.MoveDone);
		gDriver.AB[i].Wait[W_AB_UPDATEDONE]				:= BOOL_TO_DINT(gDriver.AB[i].MpAxisBasic_0.UpdateDone);
		gDriver.AB[i].Wait[W_AB_AUTOTUNEDONE]			:= BOOL_TO_DINT(gDriver.AB[i].MpAxisBasic_0.AutoTuneDone);
		gDriver.AB[i].Wait[W_AB_BRAKERELEASED]			:= BOOL_TO_DINT(gDriver.AB[i].MpAxisBasic_0.BrakeReleased);
		gDriver.AB[i].Wait[W_AB_COMMANDABORTED]			:= BOOL_TO_DINT(gDriver.AB[i].MpAxisBasic_0.CommandAborted);
		gDriver.AB[i].Wait[W_AB_COMMANDBUSY]			:= BOOL_TO_DINT(gDriver.AB[i].MpAxisBasic_0.CommandBusy);
		gDriver.AB[i].Wait[W_AB_INPOSITION]				:= BOOL_TO_DINT(gDriver.AB[i].MpAxisBasic_0.InPosition);
		gDriver.AB[i].Wait[W_AB_INVELOCITY]				:= BOOL_TO_DINT(gDriver.AB[i].MpAxisBasic_0.InVelocity);
		gDriver.AB[i].Wait[W_AB_MOVEACTIVE]				:= BOOL_TO_DINT(gDriver.AB[i].MpAxisBasic_0.MoveActive);
		gDriver.AB[i].Wait[W_AB_STOPPED]				:= BOOL_TO_DINT(gDriver.AB[i].MpAxisBasic_0.Stopped);
		gDriver.AB[i].Wait[W_AB_JOGGING]				:= BOOL_TO_DINT(gDriver.AB[i].MpAxisBasic_0.Info.Jogging);
		gDriver.AB[i].Wait[W_AB_JOGLIMITREACHED]		:= BOOL_TO_DINT(gDriver.AB[i].MpAxisBasic_0.Info.JogLimitReached);
		gDriver.AB[i].Wait[W_AB_SIMULATION]				:= BOOL_TO_DINT(gDriver.AB[i].MpAxisBasic_0.Info.Simulation);

		gDriver.AB[i].Mon[M_AB_ERROR]					:= gDriver.AB[i].MpAxisBasic_0.Error;
		gDriver.AB[i].Mon[M_AB_NOTPOWERON]				:= NOT gDriver.AB[i].MpAxisBasic_0.PowerOn;
	END_FOR;

//	McDirectionEnum :
//	(
//		mcDIR_POSITIVE := 0,							(*Movement only in the positive direction *)
//		mcDIR_NEGATIVE := 1,							(*Movement only in the negative direction*)
//		mcDIR_CURRENT := 2,								(*Movement in the direction of the active movement*)
//		mcDIR_SHORTEST_WAY := 3,						(*Movement with the shortest distance to the target, either in positive or negative direction. The movement will be in the positive direction if the distance is the same in both directions*)
//		mcDIR_EXCEED_PERIOD := 8,						(*The end position can be located outside of the axis period. The axis period can be exited in the negative direction if the end position is also negative*)
//		mcDIR_UNDEFINED := 9,							(*Movement in undefined direction*)
//		mcDIR_BOTH := 10								(*Movement in both directions*)
//	);
//	McSwitchEnum :
//	(
//		mcSWITCH_OFF := 0,		 						(*State/Behavior selection switched off*)
//		mcSWITCH_ON := 1			 					(*State/Behavior selection switched on*)
//	);
//	McHomingModeEnum :
//	(
//		mcHOMING_DIRECT := 0,							(*Direct homing. "Position" is used directly as the new axis position*)
//		mcHOMING_SWITCH_GATE := 1,						(*Homing with reference gate*)
//		mcHOMING_ABSOLUTE_SWITCH := 2,					(*Performs homing with absolute reference switch*)
//		mcHOMING_LIMIT_SWITCH := 4,	    				(*Homing with hardware limit switch*)
//		mcHOMING_ABSOLUTE := 5,							(*Homing by setting the "Position" homing offset for an absolute encoder*)
//		mcHOMING_DCM := 7,								(*Homing using interval-encoded reference marks*)
//		mcHOMING_BLOCK_TORQUE := 9,						(*Performs homing to mechanical limit, torque as criteria*)
//		mcHOMING_BLOCK_LAG_ERROR := 10,					(*Performs homing to mechanical limit, lag error as criteria*)
//		mcHOMING_ABSOLUTE_CORRECTION := 133,  			(*Homing by setting the "Position" homing offset for an absolute encoder with counter range correction. This mode must be used if the overflow of the absolute encoder is within the axis range of movement*)
//		mcHOMING_DCM_CORRECTION := 135,	 				(*Homing using distance-coded reference marks with counting range correction*)
//		mcHOMING_DEFAULT := 140,		 				(*All parameters, including "Position", are taken from the initial configuration for the axis*)
//		mcHOMING_INIT := 141,							(*All parameters, including "Position", are taken from an earlier initialization made using function block MC_BR_InitHome*)
//		mcHOMING_RESTORE_POSITION := 142				(*Restores position from a remanent variable*)
//	);
//	MpAxisAutoTuneModeEnum :
//	(
//		mcAXIS_TUNE_AUTOMATIC := 0, 					(* Performs a complete auto-tuning sequence of all controllers*)
//		mcAXIS_TUNE_SPEED := 1, 						(* Speed controller tuning*)
//		mcAXIS_TUNE_POSITION := 2, 						(* Position controller tuning*)
//		mcAXIS_TUNE_TEST := 3, 							(* Tests system stability*)
//		mcAXIS_TUNE_LOOP_FILTER := 4, 					(* Loop filter tuning*)
//		mcAXIS_TUNE_FEED_FORWARD := 5 					(*Feed forward tuning*)
//	);
//	MpAxisAutoTuneLoopFilterModeEnum :
//	(
//		mcAXIS_TUNE_LOOP_FILTER_F1 := 0, 				(*Tuning of loop filter 1 as a notch filter*)
//		mcAXIS_TUNE_LOOP_FILTER_F1_F2 := 1, 			(*Tuning of filter 1 and 2 as a notch filter*)
//		mcAXIS_TUNE_LOOP_FILTER_F1_F2_F3 := 2 			(*Tuning of filter 1, 2 and 3 as a notch filter*)
//	);
//	McAcpAxAutoTuneOrientationEnum:
//	(
//		mcACPAX_ORIENTATION_HORIZONTAL := 0, 		 	(*Horizontal orientation*)
//		mcACPAX_ORIENTATION_VERTICAL := 1    		 	(*Vertical orientation*)
//	);
//	McAcpAxFilterTimeModeEnum:
//	(
//		mcACPAX_FILTER_TIME_USE := 0,  					(*The determination of filter time constants is disabled; however, filter time constants are taken into account for autotuning*)
//		mcACPAX_FILTER_TIME_TUNE_MODE1 := 1, 		 	(*The controlled variable is the unfiltered actual speed n*)
//		mcACPAX_FILTER_TIME_TUNE_MODE2 := 2  		 	(*The controlled variable is the filtered actual speed n*)
//	);
//	McAcpAxLoopFilterModeEnum:
//	(
//		mcACPAX_LOOP_FILTER_IGNORE := 0,  				(*Loop filters are neither taken into account nor calculated.*)
//		mcACPAX_LOOP_FILTER_USE := 1,  					(*The parameters for all loop filters are taken into account for autotuning*)
//		mcACPAX_LOOP_FILTER_TUNE_NOTCH := 2  			(*The parameters for the loop filter are calculated*)
//	);
//	McAcpAxAutoTuneFeedFwdModeEnum:
//	(
//		mcACPAX_TUNE_FF_MODE_STANDARD := 0, 			(*Standard (active) tuning mode*)
//		mcACPAX_TUNE_FF_MODE_PASSIVE := 1 				(*Passive tuning mode*)
//	);
//	McAcpAxAutoTuneFeedFwdCmdEnum:
//	(
//		mcACPAX_TUNE_FF_CMD_START := 0, 				(*Start (standard or passive) tuning process*)
//		mcACPAX_TUNE_FF_CMD_FINISH := 1, 				(*Finish (passive) tuning process*)
//		mcACPAX_TUNE_FF_CMD_ABORT := 2 					(*Abort (stop) (passive) tuning process*)
//	);

END_ACTION
```

### Program Logical/Services (IEC)

#### Main.st - Init, cyclic, exit code
```iecst
PROGRAM _INIT

	gMain.Services.DirMan.In.RefreshDelay										:= 10.0;

	gMain.Services.DirMan.In.DirDef[0].Valid									:= TRUE;
	gMain.Services.DirMan.In.DirDef[0].DirPath									:= '';
	gMain.Services.DirMan.In.DirDef[0].Sanitize.AllowUndefinedDir				:= FALSE;
	gMain.Services.DirMan.In.DirDef[0].Sanitize.SanitizeFilesByRoot				:= FALSE;
	gMain.Services.DirMan.In.DirDef[0].Sanitize.SanitizeFilesByExt				:= TRUE;
	gMain.Services.DirMan.In.DirDef[0].Sanitize.FileExtension					:= '.~';
	gMain.Services.DirMan.In.DirDef[0].Sanitize.FileRoot						:= '';
	gMain.Services.DirMan.In.DirDef[0].Sanitize.MaxFiles						:= 4294967295;
	gMain.Services.DirMan.In.DirDef[0].Sanitize.MaxSize							:= 4294967295;

	gMain.Services.DirMan.In.DirDef[1].Valid									:= TRUE;
	gMain.Services.DirMan.In.DirDef[1].DirPath									:= 'Machine';
	gMain.Services.DirMan.In.DirDef[1].Sanitize.AllowUndefinedDir				:= FALSE;
	gMain.Services.DirMan.In.DirDef[1].Sanitize.SanitizeFilesByRoot				:= FALSE;
	gMain.Services.DirMan.In.DirDef[1].Sanitize.SanitizeFilesByExt				:= TRUE;
	gMain.Services.DirMan.In.DirDef[1].Sanitize.FileExtension					:= '.txt';
	gMain.Services.DirMan.In.DirDef[1].Sanitize.FileRoot						:= '';
	gMain.Services.DirMan.In.DirDef[1].Sanitize.MaxFiles						:= 4294967295;
	gMain.Services.DirMan.In.DirDef[1].Sanitize.MaxSize							:= 4294967295;

	gMain.Services.DirMan.In.DirDef[2].Valid									:= TRUE;
	gMain.Services.DirMan.In.DirDef[2].DirPath									:= 'GCODE';
	gMain.Services.DirMan.In.DirDef[2].Sanitize.AllowUndefinedDir				:= FALSE;
	gMain.Services.DirMan.In.DirDef[2].Sanitize.SanitizeFilesByRoot				:= FALSE;
	gMain.Services.DirMan.In.DirDef[2].Sanitize.SanitizeFilesByExt				:= FALSE;
	gMain.Services.DirMan.In.DirDef[2].Sanitize.FileExtension					:= '';
	gMain.Services.DirMan.In.DirDef[2].Sanitize.FileRoot						:= '';
	gMain.Services.DirMan.In.DirDef[2].Sanitize.MaxFiles						:= 100;
	gMain.Services.DirMan.In.DirDef[2].Sanitize.MaxSize							:= 4294967295;

	gMain.Services.DirMan.In.DirDef[3].Valid									:= TRUE;
	gMain.Services.DirMan.In.DirDef[3].DirPath									:= 'AlarmHistory';
	gMain.Services.DirMan.In.DirDef[3].Sanitize.AllowUndefinedDir				:= FALSE;
	gMain.Services.DirMan.In.DirDef[3].Sanitize.SanitizeFilesByRoot				:= TRUE;
	gMain.Services.DirMan.In.DirDef[3].Sanitize.SanitizeFilesByExt				:= TRUE;
	gMain.Services.DirMan.In.DirDef[3].Sanitize.FileExtension					:= '.csv';
	gMain.Services.DirMan.In.DirDef[3].Sanitize.FileRoot						:= 'Alarms';
	gMain.Services.DirMan.In.DirDef[3].Sanitize.MaxFiles						:= 10;
	gMain.Services.DirMan.In.DirDef[3].Sanitize.MaxSize							:= 4294967295;

	gMain.Services.Recipes.In.RecipeDefinitions[0].MpLink						:= gRecipeXml_Rem;
	gMain.Services.Recipes.In.RecipeDefinitions[0].DeviceName					:= gMain.Services.DeviceName;
	gMain.Services.Recipes.In.RecipeDefinitions[0].FileName						:= 'Machine/gRem.txt';
	gMain.Services.Recipes.In.RecipeDefinitions[0].VarName						:= 'gRem';
	gMain.Services.Recipes.In.RecipeDefinitions[0].pVar							:= ADR(gRem);
	gMain.Services.Recipes.In.RecipeDefinitions[0].SizeVar						:= SIZEOF(gRem);
	gMain.Services.Recipes.In.RecipeDefinitions[0].pCmpVar						:= 0;
	gMain.Services.Recipes.In.RecipeDefinitions[0].pDefaultVar					:= 0;

	gMain.Services.Recipes.In.RecipeDefinitions[1].MpLink						:= gRecipeXml_Par;
	gMain.Services.Recipes.In.RecipeDefinitions[1].DeviceName					:= gMain.Services.DeviceName;
	gMain.Services.Recipes.In.RecipeDefinitions[1].FileName						:= 'Machine/gPar.txt';
	gMain.Services.Recipes.In.RecipeDefinitions[1].VarName						:= 'gPar';
	gMain.Services.Recipes.In.RecipeDefinitions[1].pVar							:= ADR(gPar);
	gMain.Services.Recipes.In.RecipeDefinitions[1].SizeVar						:= SIZEOF(gPar);
	gMain.Services.Recipes.In.RecipeDefinitions[1].pCmpVar						:= ADR(ParCmp);
	gMain.Services.Recipes.In.RecipeDefinitions[1].pDefaultVar					:= ADR(ParDefaults);

	gMain.Services.Alarms.Internal.MpAlarmXHistoryUI_0.UISetup.AlarmListSize 	:= 50;
	gMain.Services.Alarms.Internal.MpAlarmXListUI_0.UISetup.AlarmListSize 		:= 50;

	gMain.Services.Alarms.Internal.MpAlarmXCore_0(MpLink := ADR(gAlarmXCore), Enable := TRUE, ErrorReset := gMain.ErrorReset);
	gMain.Services.Alarms.Internal.MpAlarmXListUI_0(MpLink := ADR(gAlarmXCore), Enable := TRUE, ErrorReset := gMain.ErrorReset, UIConnect := ADR(gVis.Alarms.Active.UIConnect));
	gMain.Services.Alarms.Internal.MpAlarmXHistory_0(MpLink := ADR(gAlarmXHistory), Enable := TRUE, ErrorReset := gMain.ErrorReset);
	gMain.Services.Alarms.Internal.MpAlarmXHistoryUI_0(MpLink := ADR(gAlarmXHistory), Enable := TRUE, ErrorReset := gMain.ErrorReset, UIConnect := ADR(gVis.Alarms.History.UIConnect));

END_PROGRAM

PROGRAM _CYCLIC

	Alarms;
	Recipes;
	DirMan;
	Time;

END_PROGRAM

PROGRAM _EXIT

END_PROGRAM
```

#### Variables.var - Local variables
```iecst
VAR
	ParDefaults : Par_typ;
	ParCmp : Par_typ;
	i : DINT;
END_VAR
```

#### Alarms.st
```iecst
ACTION Alarms:
	// Reactions
	gMain.Services.Alarms.Out.AlarmActive 												:= gMain.Process.Monitor.Out.SevActiveAny;
	gMain.Services.Alarms.Internal.MpAlarmXHistory_0.DeviceName 						:= ADR(gMain.Services.DeviceName);
	gMain.Services.Alarms.Internal.MpAlarmXHistory_0.FileName 							:= ADR('AlarmHistory/Alarms.csv');
	gMain.Services.Alarms.Internal.MpAlarmXHistory_0.Overwrite							:= FALSE;
	gMain.Services.Alarms.Internal.MpAlarmXHistory_0.Language							:= ADR(gPar.System.LanguageCode);
	// Case for handling the alarm history
	CASE gMain.Services.Alarms.Internal.StateExportHistory OF
		0:
			IF gMain.Services.Alarms.In.ExportHistory THEN
				TC_AlarmX_Helper(gAlarmXCore,'',TC_ALARMX_ACTION_LOG_ONLY,'HISTORY EXPORTED',FALSE);
				gMain.Services.Alarms.In.ExportHistory 									:= FALSE;
				gMain.Services.Alarms.Internal.MpAlarmXHistory_0.Export 				:= TRUE;
				gMain.Services.Alarms.Internal.StateExportHistory 						:= 10;
			ELSIF gMain.Services.Alarms.In.ClearHistory THEN
				TC_AlarmX_Helper(gAlarmXCore,'',TC_ALARMX_ACTION_LOG_ONLY,'HISTORY CLEARED',FALSE);
				gMain.Services.Alarms.In.ClearHistory 									:= FALSE;
				gMain.Services.Alarms.Internal.MpAlarmXHistory_0.Clear					:= TRUE;
			END_IF;
		10:
			IF gMain.Services.Alarms.Internal.MpAlarmXHistory_0.CommandDone OR gMain.Services.Alarms.Internal.MpAlarmXHistory_0.Error THEN
				gMain.Services.Alarms.Internal.MpAlarmXHistory_0.Export 				:= FALSE;
				gMain.Services.Alarms.Internal.StateExportHistory 						:= 0;
				gMain.Services.Alarms.Internal.MpAlarmXHistory_0.Clear					:= 0;
			END_IF;
	END_CASE;

	IF gMain.ErrorReset THEN
		gMain.Services.Alarms.In.ResetAlarms 											:= TRUE;
	END_IF;

	// Case for handling the alarm resetting
	CASE gMain.Services.Alarms.Internal.StateResetAlarms OF
		0:
			IF gMain.Services.Alarms.In.ResetAlarms OR gMain.ErrorReset THEN
				TC_AlarmX_Helper(gAlarmXCore,'',TC_ALARMX_ACTION_LOG_ONLY,'ACKNOWLEDGE ALL',FALSE);
				gMain.Services.Alarms.In.ResetAlarms 									:= FALSE;
				gVis.Alarms.Active.UIConnect.AcknowledgeAll 							:= TRUE;
				gMain.Services.Alarms.Internal.CTON_ResetDelay(IN := FALSE);
				gMain.Services.Alarms.Internal.StateResetAlarms 						:= 10;
			END_IF;
		10:
			// give UI time to process the reset
			IF gMain.Services.Alarms.Internal.CTON_ResetDelay.Q THEN
				gMain.Services.Alarms.Internal.CTON_ResetDelay(IN := FALSE);
				gMain.Services.Alarms.Internal.StateResetAlarms 						:= 0;
				gMain.ErrorReset := FALSE;
			ELSE
				gMain.Services.Alarms.Internal.CTON_ResetDelay(IN := TRUE, PT := T#250ms);
			END_IF;
	END_CASE;

	gMain.Services.Alarms.Internal.MpAlarmXListUI_0.Language							:= ADR(gPar.System.LanguageCode);

	gMain.Services.Alarms.Internal.CTON_StartDelay(IN := TRUE, PT := T#1000ms);
	IF gMain.Services.Alarms.Internal.CTON_StartDelay.Q THEN
		gMain.Services.Alarms.Out.BufferInfo.Address	:= ADR(gMain.Services.Alarms.In.AlarmList);
		gMain.Services.Alarms.Out.BufferInfo.Size		:= SIZEOF(gMain.Services.Alarms.In.AlarmList);
		gMain.Services.Alarms.Internal.TC_AlarmXCore_0.delayTime := LREAL_TO_TIME(0.5*1000.0);
		gMain.Services.Alarms.Internal.TC_AlarmXCore_0(MpLink := gAlarmXCore, enable := TRUE, pBuffer := ADR(gMain.Services.Alarms.In.AlarmList), pOutputData := ADR(gAlarmAddData));
	END_IF;
	gMain.Services.Alarms.Internal.MpAlarmXCore_0(MpLink := ADR(gAlarmXCore), Enable := TRUE, ErrorReset := gMain.ErrorReset);
	gMain.Services.Alarms.Internal.MpAlarmXListUI_0(MpLink := ADR(gAlarmXCore), Enable := TRUE, ErrorReset := gMain.ErrorReset, UIConnect := ADR(gVis.Alarms.Active.UIConnect));
	gMain.Services.Alarms.Internal.MpAlarmXHistory_0(MpLink := ADR(gAlarmXHistory), Enable := TRUE, ErrorReset := gMain.ErrorReset);
	gMain.Services.Alarms.Internal.MpAlarmXHistoryUI_0(MpLink := ADR(gAlarmXHistory), Enable := TRUE, ErrorReset := gMain.ErrorReset, UIConnect := ADR(gVis.Alarms.History.UIConnect));

END_ACTION
```

#### Defaults.st
```iecst
ACTION Defaults:

END_ACTION
```

#### Recipes.st
```iecst
ACTION Recipes:

	gMain.Services.Recipes.Out.ParametersReady 									:= TRUE;
	FOR i := 0 TO MAX_TC_RECIPE_IDX DO
		gMain.Services.Recipes.Internal.TC_Recipe_Helper_0[i](Enable := TRUE, Def := gMain.Services.Recipes.In.RecipeDefinitions[i], RemOK := gRemOK, ErrorReset := gMain.ErrorReset, ForceLoad := gMain.Services.Recipes.In.ForceLoad, ForceSave := gMain.Services.Recipes.In.ForceSave, ForceDefaults := gMain.Services.Recipes.In.ForceDefaults);
		IF NOT gMain.Services.Recipes.Internal.TC_Recipe_Helper_0[i].Initialized THEN
			gMain.Services.Recipes.Out.ParametersReady 							:= FALSE;
		END_IF;
	END_FOR;
	IF gMain.Services.Recipes.Out.ParametersReady THEN
		gRemOK																	:= TRUE;
	END_IF;
	gMain.Services.Recipes.In.ForceDefaults										:= FALSE;
	gMain.Services.Recipes.In.ForceSave											:= FALSE;
	gMain.Services.Recipes.In.ForceLoad											:= FALSE;

END_ACTION
```

#### DirMan.st
```iecst
ACTION DirMan:
	gMain.Services.DirMan.Internal.TC_Dir_USB_Connect_0.enable 							:= TRUE;

	CASE gMain.Services.DirMan.Internal.State OF
		DIR_MAN_RESET:
			gMain.Services.DirMan.In.Refresh 											:= FALSE;
			brsmemset(ADR(gMain.Services.DirMan.Out.FileList),0,SIZEOF(gMain.Services.DirMan.Out.FileList));
			brsmemset(ADR(gMain.Services.DirMan.Out.FileListUSB),0,SIZEOF(gMain.Services.DirMan.Out.FileListUSB));
			gMain.Services.DirMan.Internal.TC_DirMake_0.enable 							:= FALSE;
			gMain.Services.DirMan.Internal.TC_DirSanitize_0.enable 						:= FALSE;
			gMain.Services.DirMan.Internal.TC_Dir_USB_Connect_0.enable 					:= FALSE;
			gMain.Services.DirMan.Internal.TC_Dir_Transfer_0.enable 					:= FALSE;
			gMain.Services.DirMan.Internal.TC_DirReadAll_0.enable						:= FALSE;
			gMain.Services.DirMan.Internal.TC_DirReadAll_USB.enable						:= FALSE;
			gMain.Services.DirMan.Internal.CTON_Delay(IN := FALSE);
			gMain.Services.DirMan.Internal.State 										:= DIR_MAN_DIRMAKE_CMD;
		DIR_MAN_DIRMAKE_CMD:
			gMain.Services.DirMan.Internal.TC_DirMake_0.enable							:= TRUE;
			gMain.Services.DirMan.Internal.TC_DirMake_0.pDevice							:= ADR(gMain.Services.DeviceName);
			gMain.Services.DirMan.Internal.TC_DirMake_0.pDirDef							:= ADR(gMain.Services.DirMan.In.DirDef);
			gMain.Services.DirMan.Internal.State 										:= DIR_MAN_DIRMAKE_WAIT;
		DIR_MAN_DIRMAKE_WAIT:
			IF gMain.Services.DirMan.Internal.TC_DirMake_0.status = ERR_OK THEN
				gMain.Services.DirMan.Internal.TC_DirMake_0.enable 						:= FALSE;
				gMain.Services.DirMan.Out.DirectoriesCreated							:= TRUE;
				gMain.Services.DirMan.Internal.State 									:= DIR_MAN_DIRREAD_CMD;
			ELSIF gMain.Services.DirMan.Internal.TC_DirMake_0.status <> ERR_FUB_BUSY AND gMain.Services.DirMan.Internal.TC_DirMake_0.status <> ERR_FUB_ENABLE_FALSE THEN
				gMain.Services.DirMan.Out.DirectoriesCreated							:= FALSE;
				gMain.Services.DirMan.Internal.TC_DirMake_0.enable 						:= FALSE;
				gMain.Services.DirMan.Internal.State 									:= DIR_MAN_RESET;
			END_IF;
		DIR_MAN_DIRREAD_CMD:
			gMain.Services.DirMan.Internal.TC_DirReadAll_0.enable						:= TRUE;
			gMain.Services.DirMan.Internal.TC_DirReadAll_0.pDevice						:= ADR(gMain.Services.DeviceName);
			gMain.Services.DirMan.Internal.TC_DirReadAll_0.pFileList					:= ADR(gMain.Services.DirMan.Out.FileList);
			gMain.Services.DirMan.Internal.State 										:= DIR_MAN_DIRREAD_WAIT;
		DIR_MAN_DIRREAD_WAIT:
			IF gMain.Services.DirMan.Internal.TC_DirReadAll_0.status = ERR_OK THEN
				gMain.Services.DirMan.Internal.TC_DirReadAll_0.enable 					:= FALSE;
				gMain.Services.DirMan.Internal.State 									:= DIR_MAN_DIRREAD_USB_CMD;
			ELSIF gMain.Services.DirMan.Internal.TC_DirReadAll_0.status <> ERR_FUB_BUSY AND gMain.Services.DirMan.Internal.TC_DirReadAll_0.status <> ERR_FUB_ENABLE_FALSE THEN
				gMain.Services.DirMan.Internal.TC_DirReadAll_0.enable 					:= FALSE;
				gMain.Services.DirMan.Internal.State 									:= DIR_MAN_RESET;
			END_IF;
		DIR_MAN_DIRREAD_USB_CMD:
			IF gMain.Services.DirMan.Internal.TC_Dir_USB_Connect_0.connected THEN
				gMain.Services.DirMan.Internal.TC_DirReadAll_USB.enable					:= TRUE;
				gMain.Services.DirMan.Internal.TC_DirReadAll_USB.pDevice				:= ADR('USB_DEVICE');
				gMain.Services.DirMan.Internal.TC_DirReadAll_USB.pFileList				:= ADR(gMain.Services.DirMan.Out.FileListUSB);
				gMain.Services.DirMan.Internal.State 									:= DIR_MAN_DIRREAD_USB_WAIT;
			ELSE
				brsmemset(ADR(gMain.Services.DirMan.Out.FileListUSB),0,SIZEOF(gMain.Services.DirMan.Out.FileListUSB));
				gMain.Services.DirMan.Internal.State 									:= DIR_MAN_DIRSANITIZE_CMD;
			END_IF;
		DIR_MAN_DIRREAD_USB_WAIT:
			IF gMain.Services.DirMan.Internal.TC_DirReadAll_USB.status = ERR_OK THEN
				gMain.Services.DirMan.Internal.TC_DirReadAll_USB.enable 				:= FALSE;
				gMain.Services.DirMan.Internal.State 									:= DIR_MAN_DIRSANITIZE_CMD;
			ELSIF gMain.Services.DirMan.Internal.TC_DirReadAll_USB.status <> ERR_FUB_BUSY AND gMain.Services.DirMan.Internal.TC_DirReadAll_USB.status <> ERR_FUB_ENABLE_FALSE THEN
				gMain.Services.DirMan.Internal.TC_DirReadAll_USB.enable 				:= FALSE;
				gMain.Services.DirMan.Internal.State 									:= DIR_MAN_RESET;
			END_IF;
		DIR_MAN_DIRSANITIZE_CMD:
			gMain.Services.DirMan.Internal.TC_DirSanitize_0.enable						:= TRUE;
			gMain.Services.DirMan.Internal.TC_DirSanitize_0.pDevice						:= ADR(gMain.Services.DeviceName);
			gMain.Services.DirMan.Internal.TC_DirSanitize_0.pDirDef						:= ADR(gMain.Services.DirMan.In.DirDef);
			gMain.Services.DirMan.Internal.TC_DirSanitize_0.pFileList					:= ADR(gMain.Services.DirMan.Out.FileList);
			gMain.Services.DirMan.Internal.State 										:= DIR_MAN_DIRSANITIZE_WAIT;
		DIR_MAN_DIRSANITIZE_WAIT:
			IF gMain.Services.DirMan.Internal.TC_DirSanitize_0.status = ERR_OK THEN
				gMain.Services.DirMan.Internal.TC_DirSanitize_0.enable 					:= FALSE;
				gMain.Services.DirMan.Internal.State 									:= DIR_MAN_TRANSFER_CMD;
			ELSIF gMain.Services.DirMan.Internal.TC_DirSanitize_0.status <> ERR_FUB_BUSY AND gMain.Services.DirMan.Internal.TC_DirSanitize_0.status <> ERR_FUB_ENABLE_FALSE THEN
				gMain.Services.DirMan.Internal.TC_DirSanitize_0.enable 					:= FALSE;
				gMain.Services.DirMan.Internal.State 									:= DIR_MAN_RESET;
			END_IF;
 		DIR_MAN_TRANSFER_CMD:
			IF gMain.Services.DirMan.In.TransferList[0].Valid THEN
				gMain.Services.DirMan.Internal.TC_Dir_Transfer_0.enable 				:= TRUE;
				gMain.Services.DirMan.Internal.State 									:= DIR_MAN_TRANSFER_WAIT;
			ELSE
				gMain.Services.DirMan.Internal.TC_Dir_Transfer_0.enable 				:= FALSE;
				gMain.Services.DirMan.Internal.State 									:= DIR_MAN_DELAY;
			END_IF;
 		DIR_MAN_TRANSFER_WAIT:
			IF gMain.Services.DirMan.Internal.TC_Dir_Transfer_0.status = ERR_OK THEN
				gMain.Services.DirMan.Internal.TC_Dir_Transfer_0.enable 				:= FALSE;
				brsmemset(ADR(gMain.Services.DirMan.In.TransferList),0,SIZEOF(gMain.Services.DirMan.In.TransferList));
				gMain.Services.DirMan.In.Refresh 										:= TRUE;
				gMain.Services.DirMan.Internal.State 									:= DIR_MAN_DELAY;
			ELSIF gMain.Services.DirMan.Internal.TC_Dir_Transfer_0.status <> ERR_FUB_BUSY AND gMain.Services.DirMan.Internal.TC_Dir_Transfer_0.status <> ERR_FUB_ENABLE_FALSE THEN
				gMain.Services.DirMan.Internal.TC_Dir_Transfer_0.enable 				:= FALSE;
				gMain.Services.DirMan.Internal.State 									:= DIR_MAN_DELAY;
			END_IF;
		DIR_MAN_DELAY:
			IF gMain.Services.DirMan.Internal.CTON_Delay.Q OR gMain.Services.DirMan.In.Refresh THEN
				gMain.Services.DirMan.In.Refresh 										:= FALSE;
				gMain.Services.DirMan.Internal.CTON_Delay(IN := FALSE);
				gMain.Services.DirMan.Internal.State 									:= DIR_MAN_DIRMAKE_CMD;
			ELSIF gMain.Services.DirMan.In.TransferList[0].Valid THEN
				gMain.Services.DirMan.In.Refresh 										:= FALSE;
				gMain.Services.DirMan.Internal.CTON_Delay(IN := FALSE);
				gMain.Services.DirMan.Internal.State 									:= DIR_MAN_TRANSFER_CMD;
			ELSE
				gMain.Services.DirMan.Internal.CTON_Delay(IN := TRUE, PT := LREAL_TO_TIME(gMain.Services.DirMan.In.RefreshDelay*1000.0));
			END_IF;
	END_CASE;

	gMain.Services.DirMan.Internal.TC_DirMake_0();
	gMain.Services.DirMan.Internal.TC_DirSanitize_0();

	gMain.Services.DirMan.Internal.TC_DirReadAll_USB();
	gMain.Services.DirMan.Internal.TC_DirReadAll_0();

	gMain.Services.DirMan.Internal.TC_Dir_USB_Connect_0(delay := 0.1);
	gMain.Services.DirMan.Internal.TC_Dir_Transfer_0(USB_Connected := gMain.Services.DirMan.Internal.TC_Dir_USB_Connect_0.connected, pTransferList := ADR(gMain.Services.DirMan.In.TransferList));

END_ACTION
```

#### Time.st
```iecst
ACTION Time:

	brsmemset(ADR(gMain.Services.Time.Out), 0, SIZEOF(gMain.Services.Time.Out));

	CASE gMain.Services.Time.Internal.state OF

		TIME_RESET_C:

			gMain.Services.Time.Out.Status.CurrentState		:= 'TIME_RESET_C';
			gMain.Services.Time.Out.Status.InReset			:= TRUE;

			brsmemset(ADR(gMain.Services.Time), 0, SIZEOF(gMain.Services.Time));

			gMain.Services.Time.Internal.state				:= TIME_CHECKPARREADY_W;

		TIME_CHECKPARREADY_W:

			gMain.Services.Time.Out.Status.CurrentState		:= 'TIME_CHECKPARREADY_W';
			gMain.Services.Time.Out.Status.Initializing		:= TRUE;

			gMain.Services.Time.Internal.CTON_Timeout.PT	:= T#30s;

			IF gMain.Services.Recipes.Out.ParametersReady THEN
				gMain.Services.Time.Internal.state			:= TIME_IDLE_I;
			ELSIF gMain.Services.Time.Internal.CTON_Timeout.Q THEN
				gMain.Services.Time.Out.Status.Error		:= TRUE;
				gMain.Services.Time.Out.ErrorInfo.Severity	:= 1;
				gMain.Services.Time.Out.ErrorInfo.Text		:= 'Timeout';
				gMain.Services.Time.Out.ErrorInfo.State		:= gMain.Services.Time.Out.Status.CurrentState;
				gMain.Services.Time.Internal.state			:= TIME_ERROR;
			END_IF

		TIME_IDLE_I:

			gMain.Services.Time.Out.Status.CurrentState			:= 'TIME_IDLE_I';
			gMain.Services.Time.Out.Status.WaitingForCommand	:= TRUE;

			IF gMain.Services.Time.In.Cmd.setTime THEN
				gMain.Services.Time.In.Cmd.setTime				:= FALSE;
				gMain.Services.Time.Internal.state				:= TIME_SET_C;
			END_IF

		TIME_SET_C:

			gMain.Services.Time.Out.Status.CurrentState			:= 'TIME_SET_C';
			gMain.Services.Time.Out.Status.Processing			:= TRUE;

			gMain.Services.Time.Internal.DTSetTime_0.enable		:= TRUE;
			gMain.Services.Time.Internal.DTSetTime_0.DT1		:= gMain.Services.Time.In.Par.newTime;

			gMain.Services.Time.Internal.state					:= TIME_SET_W;

		TIME_SET_W:

			gMain.Services.Time.Out.Status.CurrentState			:= 'TIME_SET_W';
			gMain.Services.Time.Out.Status.Processing			:= TRUE;

			gMain.Services.Time.Internal.CTON_Timeout.PT		:= LREAL_TO_TIME(30.0*1000.0);

			IF gMain.Services.Time.Internal.DTSetTime_0.status = ERR_OK THEN
				gMain.Services.Time.Internal.DTSetTime_0.enable	:= FALSE;
				gMain.Services.Time.Internal.state				:= TIME_IDLE_I;
			ELSIF gMain.Services.Time.Internal.DTSetTime_0.status <> ERR_FUB_BUSY AND gMain.Services.Time.Internal.DTSetTime_0.status <> ERR_FUB_ENABLE_FALSE THEN
				gMain.Services.Time.Internal.DTSetTime_0.enable	:= FALSE;
				gMain.Services.Time.Out.ErrorInfo.Severity		:= 2;
				gMain.Services.Time.Out.ErrorInfo.Text			:= UINT_TO_STRING(gMain.Services.Time.Internal.DTSetTime_0.status);
				gMain.Services.Time.Out.ErrorInfo.State			:= gMain.Services.Time.Out.Status.CurrentState;
				gMain.Services.Time.Internal.state				:= TIME_ERROR;
			ELSIF gMain.Services.Time.Internal.CTON_Timeout.Q THEN
				gMain.Services.Time.Internal.DTSetTime_0.enable	:= FALSE;
				gMain.Services.Time.Out.ErrorInfo.Severity		:= 2;
				gMain.Services.Time.Out.ErrorInfo.Text			:= 'Timeout';
				gMain.Services.Time.Out.ErrorInfo.State			:= gMain.Services.Time.Out.Status.CurrentState;
				gMain.Services.Time.Internal.state				:= TIME_ERROR;
			END_IF

		TIME_ERROR:

			gMain.Services.Time.Out.Status.CurrentState			:= 'TIME_ERROR';
			gMain.Services.Time.Out.Status.InError				:= TRUE;

			IF gMain.ErrorReset THEN
				gMain.Services.Time.Internal.state				:= TIME_RESET_C;
			END_IF

	END_CASE;

	//Update Current Time output

	gMain.Services.Time.Out.Status.CurrentTime 		:= gMain.Services.Time.Internal.DTGetTime_0.DT1;

	IF gMain.Services.Time.Out.Status.CurrentTime > DT#2024-01-01-00:00:00 THEN
		gMain.Services.Time.Out.Status.TimeValid	:= TRUE;
	END_IF

	IF NOT gMain.Services.Time.Out.Status.WaitingForCommand THEN
		IF gMain.Services.Time.In.Cmd.setTime THEN
			gMain.Services.Time.In.Cmd.setTime												:= FALSE;
			gMain.Services.Time.Out.IgnoreInfo.Cmd											:= 'Set Time';
			gMain.Services.Time.Out.IgnoreInfo.Reason										:= 'Not in Waiting for Command';
			gMain.Services.Time.Out.ErrorInfo.State											:= gMain.Services.Time.Out.Status.CurrentState;
			TC_AlarmX_Helper(gAlarmXCore,'TimeCmdIgnored',TC_ALARMX_ACTION_SET,'',TRUE);
		END_IF;
	END_IF;
	brsmemset(ADR(gMain.Services.Time.Internal.BlankCmdCmp),0,SIZEOF(gMain.Services.Time.Internal.BlankCmdCmp));
	IF brsmemcmp(ADR(gMain.Services.Time.Internal.BlankCmdCmp),ADR(gMain.Services.Time.In.Cmd),SIZEOF(gMain.Services.Time.In.Cmd)) <> 0 THEN
		gMain.Services.Time.Out.ErrorInfo.State													:= gMain.Services.Time.Out.Status.CurrentState;
		TC_AlarmX_Helper(gAlarmXCore,'TimeUnhandledCmd',TC_ALARMX_ACTION_SET,'',TRUE);
	END_IF;
	brsmemset(ADR(gMain.Services.Time.In.Cmd),0,SIZEOF(gMain.Services.Time.In.Cmd));

	IF gMain.Services.Time.Out.Status.Error THEN
		IF brsmemcmp(ADR(gMain.Services.Time.Internal.LastErrorInfo),ADR(gMain.Services.Time.Out.ErrorInfo),SIZEOF(gMain.Services.Time.Internal.LastErrorInfo)) <> 0 THEN
			brsmemcpy(ADR(gMain.Services.Time.Internal.LastErrorInfo),ADR(gMain.Services.Time.Out.ErrorInfo),SIZEOF(gMain.Services.Time.Internal.LastErrorInfo));
			CASE gMain.Services.Time.Out.ErrorInfo.Severity OF
				1:
					gMain.Services.Time.Internal.tempAlarm.name				:= 'TimeSeverity1';
					gMain.Services.Time.Internal.tempAlarm.allowMultiple		:= TRUE;
					gMain.Services.Time.Internal.tempAlarm.addText[0]			:= gMain.Services.Time.Out.ErrorInfo.State;
					gMain.Services.Time.Internal.tempAlarm.addText[1]			:= gMain.Services.Time.Out.ErrorInfo.Text;

					TC_Array_AddTop(ADR(gMain.Services.Alarms.In.AlarmList), SIZEOF(gMain.Services.Alarms.In.AlarmList), ADR(gMain.Services.Time.Internal.tempAlarm), SIZEOF(gMain.Services.Time.Internal.tempAlarm));
				2:
					gMain.Services.Time.Internal.tempAlarm.name				:= 'TimeSeverity2';
					gMain.Services.Time.Internal.tempAlarm.allowMultiple		:= TRUE;
					gMain.Services.Time.Internal.tempAlarm.addText[0]			:= gMain.Services.Time.Out.ErrorInfo.State;
					gMain.Services.Time.Internal.tempAlarm.addText[1]			:= gMain.Services.Time.Out.ErrorInfo.Text;
					brsitoa(gMain.Services.Time.Out.ErrorInfo.Code, ADR(gMain.Services.Time.Internal.tempAlarm.addText[2]));

					TC_Array_AddTop(ADR(gMain.Services.Alarms.In.AlarmList), SIZEOF(gMain.Services.Alarms.In.AlarmList), ADR(gMain.Services.Time.Internal.tempAlarm), SIZEOF(gMain.Services.Time.Internal.tempAlarm));
				3:
					gMain.Services.Time.Internal.tempAlarm.name				:= 'TimeSeverity3';
					gMain.Services.Time.Internal.tempAlarm.allowMultiple		:= TRUE;
					gMain.Services.Time.Internal.tempAlarm.addText[0]			:= gMain.Services.Time.Out.ErrorInfo.State;
					gMain.Services.Time.Internal.tempAlarm.addText[1]			:= gMain.Services.Time.Out.ErrorInfo.Text;

					TC_Array_AddTop(ADR(gMain.Services.Alarms.In.AlarmList), SIZEOF(gMain.Services.Alarms.In.AlarmList), ADR(gMain.Services.Time.Internal.tempAlarm), SIZEOF(gMain.Services.Time.Internal.tempAlarm));
				4:
					gMain.Services.Time.Internal.tempAlarm.name				:= 'TimeSeverity4';
					gMain.Services.Time.Internal.tempAlarm.allowMultiple		:= TRUE;
					gMain.Services.Time.Internal.tempAlarm.addText[0]			:= gMain.Services.Time.Out.ErrorInfo.State;
					gMain.Services.Time.Internal.tempAlarm.addText[1]			:= gMain.Services.Time.Out.ErrorInfo.Text;

					TC_Array_AddTop(ADR(gMain.Services.Alarms.In.AlarmList), SIZEOF(gMain.Services.Alarms.In.AlarmList), ADR(gMain.Services.Time.Internal.tempAlarm), SIZEOF(gMain.Services.Time.Internal.tempAlarm));
			END_CASE;
		END_IF;
	ELSE
		brsmemset(ADR(gMain.Services.Time.Internal.LastErrorInfo),0,SIZEOF(gMain.Services.Time.Internal.LastErrorInfo));
	END_IF;

	//Reset Timers on state change
	IF gMain.Services.Time.Internal.lastState <> gMain.Services.Time.Internal.state OR gMain.Services.Time.Internal.state = TIME_RESET_C THEN
		gMain.Services.Time.Internal.lastState													:= gMain.Services.Time.Internal.state;
		gMain.Services.Time.Internal.CTON_Timeout.IN											:= FALSE;
		gMain.Services.Time.Internal.CTON_Delay.IN												:= FALSE;
	END_IF;

	//Function Calls
	gMain.Services.Time.Internal.CTON_Timeout(PAUSE := FALSE);
	gMain.Services.Time.Internal.CTON_Delay(PAUSE := FALSE);
	gMain.Services.Time.Internal.DTGetTime_0(enable:=TRUE);
	gMain.Services.Time.Internal.DTSetTime_0();

END_ACTION
```

#### Cert.st - not listed in the package file held
```iecst
ACTION Cert:

	gMain.Services.Cert.In.Par.CountryCode														:= gPar.Services.Cert.CountryCode;
	gMain.Services.Cert.In.Par.StateProvince													:= gPar.Services.Cert.StateProvince;
	gMain.Services.Cert.In.Par.Locality															:= gPar.Services.Cert.Locality;
	gMain.Services.Cert.In.Par.Organization														:= gPar.Services.Cert.Organization;
	gMain.Services.Cert.In.Par.OrganizationUnit													:= gPar.Services.Cert.OrganizationUnit;
	gMain.Services.Cert.In.Par.ContactEmail														:= gPar.Services.Cert.ContactEmail;
	gMain.Services.Cert.In.Par.CommonName														:= gPar.Services.Cert.CommonName;
	gMain.Services.Cert.In.Par.IP																:= gPar.Services.Cert.IP;

	IF gMain.Services.Cert.In.Cmd.Reset THEN
		gMain.Services.Cert.In.Cmd.Reset														:= FALSE;
		gMain.Services.Cert.Internal.State														:= CERT_RESET_C;
	END_IF;

	brsmemset(ADR(gMain.Services.Cert.Out),0,SIZEOF(gMain.Services.Cert.Out));
	CASE gMain.Services.Cert.Internal.State OF
		CERT_RESET_C:
			gMain.Services.Cert.Out.Status.CurrentState											:= 'CERT_RESET_C';
			gMain.Services.Cert.Out.Status.InReset												:= TRUE;
			brsmemset(ADR(gMain.Services.Cert.In),0,SIZEOF(gMain.Services.Cert.In));
			brsmemset(ADR(gMain.Services.Cert.Internal),0,SIZEOF(gMain.Services.Cert.Internal));
			gMain.Services.Cert.Internal.State 													:= CERT_CHECKPARREADY_W;
		CERT_CHECKPARREADY_W:
			gMain.Services.Cert.Out.Status.CurrentState											:= 'CERT_CHECKPARREADY_W';
			gMain.Services.Cert.Out.Status.Initializing											:= TRUE;
			gMain.Services.Cert.Internal.CTON_Timeout.IN 										:= TRUE;
			gMain.Services.Cert.Internal.CTON_Timeout.PT 										:= LREAL_TO_TIME(30.0*1000.0); //Hardcoded because parameters are not yet loaded
			IF gMain.Services.Recipes.Out.ParametersReady THEN
				gMain.Services.Cert.Internal.State 												:= CERT_IDLE_I;
			ELSIF gMain.Services.Cert.Internal.CTON_Timeout.Q THEN
				gMain.Services.Cert.Out.Status.Error 											:= TRUE;
				gMain.Services.Cert.Out.ErrorInfo.Severity										:= 1;
				gMain.Services.Cert.Out.ErrorInfo.Text 											:= 'Timeout';
				gMain.Services.Cert.Out.ErrorInfo.State 										:= gMain.Services.Cert.Out.Status.CurrentState;
				gMain.Services.Cert.Internal.State 												:= CERT_ERROR_I;
			END_IF;
		CERT_IDLE_I:
			gMain.Services.Cert.Out.Status.CurrentState											:= 'CERT_IDLE_I';
			gMain.Services.Cert.Out.Status.WaitingForCommand									:= TRUE;
			IF gMain.Services.Cert.SSLConfigIdent = 0 THEN
				gMain.Services.Cert.Internal.State 												:= CERT_GEN_CERT_D;
			END_IF;
		CERT_GEN_CERT_D:
			gMain.Services.Cert.Out.Status.CurrentState											:= 'CERT_GEN_CERT_D';
			gMain.Services.Cert.Out.Status.Processing											:= TRUE;
			gMain.Services.Cert.Internal.CTON_Delay.IN 											:= TRUE;
			gMain.Services.Cert.Internal.CTON_Delay.PT 											:= LREAL_TO_TIME(0.0*1000.0);
			IF gMain.Services.Cert.Internal.CTON_Delay.Q OR 0.0 < 0.0001 THEN
				gMain.Services.Cert.Internal.State 												:= CERT_GEN_CERT_C;
			END_IF;
		CERT_GEN_CERT_C:
			gMain.Services.Cert.Out.Status.CurrentState											:= 'CERT_GEN_CERT_C';
			gMain.Services.Cert.Out.Status.Processing											:= TRUE;
			gMain.Services.Cert.Internal.ArCertGenerateX_0.Execute								:= TRUE;
			gMain.Services.Cert.Internal.ArCertGenerateX_0.Name									:= 'AutoGenerated.cer';
			gMain.Services.Cert.Internal.ArCertGenerateX_0.PrivateKeyName						:= 'AutoGenerated.key';
			gMain.Services.Cert.Internal.ArCertGenerateX_0.CountryCode							:= gMain.Services.Cert.In.Par.CountryCode;
			gMain.Services.Cert.Internal.ArCertGenerateX_0.StateProvince						:= gMain.Services.Cert.In.Par.StateProvince;
			gMain.Services.Cert.Internal.ArCertGenerateX_0.Locality								:= gMain.Services.Cert.In.Par.Locality;
			gMain.Services.Cert.Internal.ArCertGenerateX_0.Organization						   	:= gMain.Services.Cert.In.Par.Organization;
			gMain.Services.Cert.Internal.ArCertGenerateX_0.OrganizationUnit						:= gMain.Services.Cert.In.Par.OrganizationUnit;
			gMain.Services.Cert.Internal.ArCertGenerateX_0.ContactEmail							:= gMain.Services.Cert.In.Par.ContactEmail;
			gMain.Services.Cert.Internal.ArCertGenerateX_0.CommonName							:= gMain.Services.Cert.In.Par.CommonName;
			gMain.Services.Cert.Internal.ArCertGenerateX_0.IP									:= gMain.Services.Cert.In.Par.IP;
			gMain.Services.Cert.Internal.ArCertGenerateX_0.KeySize								:= arCERT_KEY_SIZE_4096_BITS;
			gMain.Services.Cert.Internal.ArCertGenerateX_0.ValidTimeSeconds						:= 365*24*60*60; // 1 year
			gMain.Services.Cert.Internal.ArCertGenerateX_0.DnsName								:= '';
			gMain.Services.Cert.Internal.ArCertGenerateX_0.URI									:= 'urn:';
			TC_brsstrcat(ADR(gMain.Services.Cert.Internal.ArCertGenerateX_0.URI),ADR(gMain.Services.Cert.In.Par.IP),SIZEOF(gMain.Services.Cert.Internal.ArCertGenerateX_0.URI));
			TC_brsstrcat(ADR(gMain.Services.Cert.Internal.ArCertGenerateX_0.URI),ADR('/BR/'),SIZEOF(gMain.Services.Cert.Internal.ArCertGenerateX_0.URI));
			gMain.Services.Cert.Internal.State 													:= CERT_GEN_CERT_W;
		CERT_GEN_CERT_W:
			gMain.Services.Cert.Out.Status.CurrentState											:= 'CERT_GEN_CERT_W';
			gMain.Services.Cert.Out.Status.Processing											:= TRUE;
			gMain.Services.Cert.Internal.CTON_Timeout.IN 										:= TRUE;
			gMain.Services.Cert.Internal.CTON_Timeout.PT 										:= LREAL_TO_TIME(30.0*1000.0);
			IF gMain.Services.Cert.Internal.ArCertGenerateX_0.StatusID = 0 AND gMain.Services.Cert.Internal.ArCertGenerateX_0.Done THEN
				gMain.Services.Cert.Internal.ArCertGenerateX_0.Execute							:= FALSE;
				gMain.Services.Cert.Internal.State 												:= CERT_DELETE_SSL_D;
			ELSIF gMain.Services.Cert.Internal.ArCertGenerateX_0.Error OR (gMain.Services.Cert.Internal.ArCertGenerateX_0.StatusID <> 0 AND gMain.Services.Cert.Internal.ArCertGenerateX_0.StatusID <> 65535 AND gMain.Services.Cert.Internal.ArCertGenerateX_0.StatusID <> 65534) THEN
				gMain.Services.Cert.Internal.ArCertGenerateX_0.Execute							:= FALSE;
				gMain.Services.Cert.Out.Status.Error 											:= TRUE;
				gMain.Services.Cert.Out.ErrorInfo.Severity										:= 2;
				gMain.Services.Cert.Out.ErrorInfo.Code 											:= gMain.Services.Cert.Internal.ArCertGenerateX_0.StatusID;
				gMain.Services.Cert.Out.ErrorInfo.Text 											:= 'FBError';
				gMain.Services.Cert.Internal.State 												:= CERT_ERROR_I;
			ELSIF gMain.Services.Cert.Internal.CTON_Timeout.Q THEN
				gMain.Services.Cert.Internal.ArCertGenerateX_0.Execute							:= FALSE;
				gMain.Services.Cert.Out.Status.Error 											:= TRUE;
				gMain.Services.Cert.Out.ErrorInfo.Severity										:= 2;
				gMain.Services.Cert.Out.ErrorInfo.Text 											:= 'Timeout';
				gMain.Services.Cert.Internal.State 												:= CERT_ERROR_I;
			END_IF;
		CERT_DELETE_SSL_D:
			gMain.Services.Cert.Out.Status.CurrentState											:= 'CERT_DELETE_SSL_D';
			gMain.Services.Cert.Out.Status.Processing											:= TRUE;
			gMain.Services.Cert.Internal.CTON_Delay.IN 											:= TRUE;
			gMain.Services.Cert.Internal.CTON_Delay.PT 											:= LREAL_TO_TIME(0.0*1000.0);
			IF gMain.Services.Cert.Internal.CTON_Delay.Q OR 0.0 < 0.0001 THEN
				gMain.Services.Cert.Internal.State 												:= CERT_DELETE_SSL_C;
			END_IF;
		CERT_DELETE_SSL_C:
			gMain.Services.Cert.Out.Status.CurrentState											:= 'CERT_DELETE_SSL_C';
			gMain.Services.Cert.Out.Status.Processing											:= TRUE;
			gMain.Services.Cert.Internal.ArSslDeleteCfg_0.Execute								:= TRUE;
			gMain.Services.Cert.Internal.ArSslDeleteCfg_0.Name									:= 'AutoGenerated';
			gMain.Services.Cert.Internal.State 													:= CERT_DELETE_SSL_W;
		CERT_DELETE_SSL_W:
			gMain.Services.Cert.Out.Status.CurrentState											:= 'CERT_DELETE_SSL_W';
			gMain.Services.Cert.Out.Status.Processing											:= TRUE;
			gMain.Services.Cert.Internal.CTON_Timeout.IN 										:= TRUE;
			gMain.Services.Cert.Internal.CTON_Timeout.PT 										:= LREAL_TO_TIME(30.0*1000.0);
			IF (gMain.Services.Cert.Internal.ArSslDeleteCfg_0.Done OR gMain.Services.Cert.Internal.ArSslDeleteCfg_0.Error) AND (gMain.Services.Cert.Internal.ArSslDeleteCfg_0.StatusID = 0 OR gMain.Services.Cert.Internal.ArSslDeleteCfg_0.StatusID = arSSL_ERR_SSL_CFG_NOT_FOUND) THEN
				gMain.Services.Cert.Internal.ArSslDeleteCfg_0.Execute							:= FALSE;
				gMain.Services.Cert.Internal.State 												:= CERT_CREATE_SSL_D;
			ELSIF gMain.Services.Cert.Internal.ArSslDeleteCfg_0.Error OR (gMain.Services.Cert.Internal.ArSslDeleteCfg_0.StatusID <> 0 AND gMain.Services.Cert.Internal.ArSslDeleteCfg_0.StatusID <> arSSL_ERR_SSL_CFG_NOT_FOUND AND gMain.Services.Cert.Internal.ArSslDeleteCfg_0.StatusID <> 65535 AND gMain.Services.Cert.Internal.ArSslDeleteCfg_0.StatusID <> 65534) THEN
				gMain.Services.Cert.Internal.ArSslDeleteCfg_0.Execute							:= FALSE;
				gMain.Services.Cert.Out.Status.Error 											:= TRUE;
				gMain.Services.Cert.Out.ErrorInfo.Severity										:= 2;
				gMain.Services.Cert.Out.ErrorInfo.Code 											:= gMain.Services.Cert.Internal.ArSslDeleteCfg_0.StatusID;
				gMain.Services.Cert.Out.ErrorInfo.Text 											:= 'FBError';
				gMain.Services.Cert.Internal.State 												:= CERT_ERROR_I;
			ELSIF gMain.Services.Cert.Internal.CTON_Timeout.Q THEN
				gMain.Services.Cert.Internal.ArSslDeleteCfg_0.Execute							:= FALSE;
				gMain.Services.Cert.Out.Status.Error 											:= TRUE;
				gMain.Services.Cert.Out.ErrorInfo.Severity										:= 2;
				gMain.Services.Cert.Out.ErrorInfo.Text 											:= 'Timeout';
				gMain.Services.Cert.Internal.State 												:= CERT_ERROR_I;
			END_IF;
		CERT_CREATE_SSL_D:
			gMain.Services.Cert.Out.Status.CurrentState											:= 'CERT_CREATE_SSL_D';
			gMain.Services.Cert.Out.Status.Processing											:= TRUE;
			gMain.Services.Cert.Internal.CTON_Delay.IN 											:= TRUE;
			gMain.Services.Cert.Internal.CTON_Delay.PT 											:= LREAL_TO_TIME(0.0*1000.0);
			IF gMain.Services.Cert.Internal.CTON_Delay.Q OR 0.0 < 0.0001 THEN
				gMain.Services.Cert.Internal.State 												:= CERT_CREATE_SSL_C;
			END_IF;
		CERT_CREATE_SSL_C:
			gMain.Services.Cert.Out.Status.CurrentState												:= 'CERT_CREATE_SSL_C';
			gMain.Services.Cert.Out.Status.Processing												:= TRUE;
			gMain.Services.Cert.Internal.ArSslCreateCfg_0.Execute									:= TRUE;
			gMain.Services.Cert.Internal.ArSslCreateCfg_0.Name										:= 'AutoGenerated';
			gMain.Services.Cert.Internal.ArSslCreateCfg_0.Configuration.OwnCertificate.Certificate	:= 'AutoGenerated.cer';
			gMain.Services.Cert.Internal.ArSslCreateCfg_0.Configuration.OwnCertificate.PrivateKey	:= 'AutoGenerated.key';
			gMain.Services.Cert.Internal.ArSslCreateCfg_0.Configuration.OwnCertificate.Password		:= '';
			gMain.Services.Cert.Internal.ArSslCreateCfg_0.Configuration.SslVersion					:= arSSL_TLS_1_2;
			gMain.Services.Cert.Internal.ArSslCreateCfg_0.Configuration.CRLCount					:= 0;
			gMain.Services.Cert.Internal.ArSslCreateCfg_0.Configuration.CRLs						:= 0;
			gMain.Services.Cert.Internal.ArSslCreateCfg_0.Configuration.TrustedCertificateCount		:= 0;
			gMain.Services.Cert.Internal.ArSslCreateCfg_0.Configuration.TrustedCertificates			:= 0;
			gMain.Services.Cert.Internal.State 														:= CERT_CREATE_SSL_W;
		CERT_CREATE_SSL_W:
			gMain.Services.Cert.Out.Status.CurrentState											:= 'CERT_CREATE_SSL_W';
			gMain.Services.Cert.Out.Status.Processing											:= TRUE;
			gMain.Services.Cert.Internal.CTON_Timeout.IN 										:= TRUE;
			gMain.Services.Cert.Internal.CTON_Timeout.PT 										:= LREAL_TO_TIME(30.0*1000.0);
			IF gMain.Services.Cert.Internal.ArSslCreateCfg_0.Done AND gMain.Services.Cert.Internal.ArSslCreateCfg_0.StatusID = 0 THEN
				gMain.Services.Cert.Internal.ArSslCreateCfg_0.Execute							:= FALSE;
				gMain.Services.Cert.Internal.State 												:= CERT_OPEN_SSL_D;
			ELSIF gMain.Services.Cert.Internal.ArSslCreateCfg_0.Error OR (gMain.Services.Cert.Internal.ArSslCreateCfg_0.StatusID <> 0 AND gMain.Services.Cert.Internal.ArSslCreateCfg_0.StatusID <> 65535 AND gMain.Services.Cert.Internal.ArSslCreateCfg_0.StatusID <> 65534) THEN
				gMain.Services.Cert.Internal.ArSslCreateCfg_0.Execute							:= FALSE;
				gMain.Services.Cert.Out.Status.Error 											:= TRUE;
				gMain.Services.Cert.Out.ErrorInfo.Severity										:= 2;
				gMain.Services.Cert.Out.ErrorInfo.Code 											:= gMain.Services.Cert.Internal.ArSslCreateCfg_0.StatusID;
				gMain.Services.Cert.Out.ErrorInfo.Text 											:= 'FBError';
				gMain.Services.Cert.Internal.State 												:= CERT_ERROR_I;
			ELSIF gMain.Services.Cert.Internal.CTON_Timeout.Q THEN
				gMain.Services.Cert.Internal.ArSslCreateCfg_0.Execute							:= FALSE;
				gMain.Services.Cert.Out.Status.Error 											:= TRUE;
				gMain.Services.Cert.Out.ErrorInfo.Severity										:= 2;
				gMain.Services.Cert.Out.ErrorInfo.Text 											:= 'Timeout';
				gMain.Services.Cert.Internal.State 												:= CERT_ERROR_I;
			END_IF;
		CERT_OPEN_SSL_D:
			gMain.Services.Cert.Out.Status.CurrentState											:= 'CERT_OPEN_SSL_D';
			gMain.Services.Cert.Out.Status.Processing											:= TRUE;
			gMain.Services.Cert.Internal.CTON_Delay.IN 											:= TRUE;
			gMain.Services.Cert.Internal.CTON_Delay.PT 											:= LREAL_TO_TIME(0.0*1000.0);
			IF gMain.Services.Cert.Internal.CTON_Delay.Q OR 0.0 < 0.0001 THEN
				gMain.Services.Cert.Internal.State 												:= CERT_OPEN_SSL_C;
			END_IF;
		CERT_OPEN_SSL_C:
			gMain.Services.Cert.Out.Status.CurrentState											:= 'CERT_OPEN_SSL_C';
			gMain.Services.Cert.Out.Status.Processing											:= TRUE;
			gMain.Services.Cert.Internal.ArSslOpen_0.Execute									:= TRUE;
			gMain.Services.Cert.Internal.ArSslOpen_0.Name										:= 'AutoGenerated';
			gMain.Services.Cert.Internal.State 													:= CERT_OPEN_SSL_W;
		CERT_OPEN_SSL_W:
			gMain.Services.Cert.Out.Status.CurrentState											:= 'CERT_OPEN_SSL_W';
			gMain.Services.Cert.Out.Status.Processing											:= TRUE;
			gMain.Services.Cert.Internal.CTON_Timeout.IN 										:= TRUE;
			gMain.Services.Cert.Internal.CTON_Timeout.PT 										:= LREAL_TO_TIME(30.0*1000.0);

			IF gMain.Services.Cert.Internal.ArSslOpen_0.Done AND gMain.Services.Cert.Internal.ArSslOpen_0.StatusID = 0 THEN
				gMain.Services.Cert.Internal.ArSslOpen_0.Execute								:= FALSE;
				gMain.Services.Cert.SSLConfigIdent												:= gMain.Services.Cert.Internal.ArSslOpen_0.Ident;
				gMain.Services.Cert.Internal.State 												:= CERT_IDLE_I;
			ELSIF gMain.Services.Cert.Internal.ArSslOpen_0.Error OR (gMain.Services.Cert.Internal.ArSslOpen_0.StatusID <> 0 AND gMain.Services.Cert.Internal.ArSslOpen_0.StatusID <> 65535 AND gMain.Services.Cert.Internal.ArSslOpen_0.StatusID <> 65534) THEN
				gMain.Services.Cert.Internal.ArSslOpen_0.Execute								:= FALSE;
				gMain.Services.Cert.Out.Status.Error 											:= TRUE;
				gMain.Services.Cert.Out.ErrorInfo.Severity										:= 2;
				gMain.Services.Cert.Out.ErrorInfo.Code 											:= gMain.Services.Cert.Internal.ArSslOpen_0.StatusID;
				gMain.Services.Cert.Out.ErrorInfo.Text 											:= 'FBError';
				gMain.Services.Cert.Internal.State 												:= CERT_ERROR_I;
			ELSIF gMain.Services.Cert.Internal.CTON_Timeout.Q THEN
				gMain.Services.Cert.Internal.ArSslOpen_0.Execute								:= FALSE;
				gMain.Services.Cert.Out.Status.Error 											:= TRUE;
				gMain.Services.Cert.Out.ErrorInfo.Severity										:= 2;
				gMain.Services.Cert.Out.ErrorInfo.Text 											:= 'Timeout';
				gMain.Services.Cert.Internal.State 												:= CERT_ERROR_I;
			END_IF;
		CERT_ERROR_I:
			gMain.Services.Cert.Out.Status.CurrentState											:= 'CERT_ERROR_I';
			gMain.Services.Cert.Out.Status.InError 												:= TRUE;
			gMain.Services.Cert.SSLConfigIdent													:= 0;
			IF gMain.ErrorReset THEN
				gMain.Services.Cert.Internal.State 												:= CERT_RESET_C;
			END_IF;
	END_CASE;
	//Check for Commands that are still true. If they are still true then they were not handled and we need to error.
	brsmemset(ADR(gMain.Services.Cert.Internal.BlankCmdCmp),0,SIZEOF(gMain.Services.Cert.Internal.BlankCmdCmp));
	IF brsmemcmp(ADR(gMain.Services.Cert.Internal.BlankCmdCmp),ADR(gMain.Services.Cert.In.Cmd),SIZEOF(gMain.Services.Cert.In.Cmd)) <> 0 THEN
		gMain.Services.Cert.Out.ErrorInfo.State												:= gMain.Services.Cert.Out.Status.CurrentState;

		gMain.Services.Cert.Internal.tempAlarm.name											:= 'CertUnhandledCmd';
		gMain.Services.Cert.Internal.tempAlarm.allowMultiple									:= TRUE;
		gMain.Services.Cert.Internal.tempAlarm.addText[0]										:= gMain.Services.Cert.Out.ErrorInfo.State;
		TC_Array_AddTop(ADR(gMain.Services.Alarms.In.AlarmList), SIZEOF(gMain.Services.Alarms.In.AlarmList), ADR(gMain.Services.Cert.Internal.tempAlarm), SIZEOF(gMain.Services.Cert.Internal.tempAlarm));
	END_IF;
	brsmemset(ADR(gMain.Services.Cert.In.Cmd),0,SIZEOF(gMain.Services.Cert.In.Cmd));

	//Reset Timeout On State Change
	IF gMain.Services.Cert.Internal.LastState <> gMain.Services.Cert.Internal.State OR gMain.Services.Cert.Internal.State = CERT_RESET_C THEN
		gMain.Services.Cert.Internal.LastState													:= gMain.Services.Cert.Internal.State;
		gMain.Services.Cert.Internal.CTON_Timeout.IN											:= FALSE;
		gMain.Services.Cert.Internal.CTON_Delay.IN												:= FALSE;
	END_IF;

	//Function Calls
	gMain.Services.Cert.Internal.CTON_Timeout(PAUSE := FALSE);
	gMain.Services.Cert.Internal.CTON_Delay(PAUSE := FALSE);
	gMain.Services.Cert.Internal.ArCertGenerateX_0();
	gMain.Services.Cert.Internal.ArSslCreateCfg_0();
	gMain.Services.Cert.Internal.ArSslDeleteCfg_0();
	gMain.Services.Cert.Internal.ArSslOpen_0();

	//Error Collection
	IF gMain.Services.Cert.Out.Status.Error THEN
		IF brsmemcmp(ADR(gMain.Services.Cert.Internal.LastErrorInfo),ADR(gMain.Services.Cert.Out.ErrorInfo),SIZEOF(gMain.Services.Cert.Internal.LastErrorInfo)) <> 0 THEN
			brsmemcpy(ADR(gMain.Services.Cert.Internal.LastErrorInfo),ADR(gMain.Services.Cert.Out.ErrorInfo),SIZEOF(gMain.Services.Cert.Internal.LastErrorInfo));
			CASE gMain.Services.Cert.Out.ErrorInfo.Severity OF
				1:
					gMain.Services.Cert.Internal.tempAlarm.name				:= 'CertSeverity1';
					gMain.Services.Cert.Internal.tempAlarm.allowMultiple		:= TRUE;
					gMain.Services.Cert.Internal.tempAlarm.addText[0]			:= gMain.Services.Cert.Out.ErrorInfo.State;
					gMain.Services.Cert.Internal.tempAlarm.addText[1]			:= gMain.Services.Cert.Out.ErrorInfo.Text;

					TC_Array_AddTop(ADR(gMain.Services.Alarms.In.AlarmList), SIZEOF(gMain.Services.Alarms.In.AlarmList), ADR(gMain.Services.Cert.Internal.tempAlarm), SIZEOF(gMain.Services.Cert.Internal.tempAlarm));
				2:
					gMain.Services.Cert.Internal.tempAlarm.name				:= 'CertSeverity2';
					gMain.Services.Cert.Internal.tempAlarm.allowMultiple		:= TRUE;
					gMain.Services.Cert.Internal.tempAlarm.addText[0]			:= gMain.Services.Cert.Out.ErrorInfo.State;
					gMain.Services.Cert.Internal.tempAlarm.addText[1]			:= gMain.Services.Cert.Out.ErrorInfo.Text;
					gMain.Services.Cert.Internal.tempAlarm.addText[2]			:= DINT_TO_STRING(gMain.Services.Cert.Out.ErrorInfo.Code);
					brsitoa(gMain.Services.Cert.Out.ErrorInfo.Code, ADR(gMain.Services.Cert.Internal.tempAlarm.addText[2]));

					TC_Array_AddTop(ADR(gMain.Services.Alarms.In.AlarmList), SIZEOF(gMain.Services.Alarms.In.AlarmList), ADR(gMain.Services.Cert.Internal.tempAlarm), SIZEOF(gMain.Services.Cert.Internal.tempAlarm));
				3:
					gMain.Services.Cert.Internal.tempAlarm.name				:= 'CertSeverity3';
					gMain.Services.Cert.Internal.tempAlarm.allowMultiple		:= TRUE;
					gMain.Services.Cert.Internal.tempAlarm.addText[0]			:= gMain.Services.Cert.Out.ErrorInfo.State;
					gMain.Services.Cert.Internal.tempAlarm.addText[1]			:= gMain.Services.Cert.Out.ErrorInfo.Text;

					TC_Array_AddTop(ADR(gMain.Services.Alarms.In.AlarmList), SIZEOF(gMain.Services.Alarms.In.AlarmList), ADR(gMain.Services.Cert.Internal.tempAlarm), SIZEOF(gMain.Services.Cert.Internal.tempAlarm));
				4:
					gMain.Services.Cert.Internal.tempAlarm.name				:= 'CertSeverity4';
					gMain.Services.Cert.Internal.tempAlarm.allowMultiple		:= TRUE;
					gMain.Services.Cert.Internal.tempAlarm.addText[0]			:= gMain.Services.Cert.Out.ErrorInfo.State;
					gMain.Services.Cert.Internal.tempAlarm.addText[1]			:= gMain.Services.Cert.Out.ErrorInfo.Text;

					TC_Array_AddTop(ADR(gMain.Services.Alarms.In.AlarmList), SIZEOF(gMain.Services.Alarms.In.AlarmList), ADR(gMain.Services.Cert.Internal.tempAlarm), SIZEOF(gMain.Services.Cert.Internal.tempAlarm));
			END_CASE;
		END_IF;
	ELSE
		brsmemset(ADR(gMain.Services.Cert.Internal.LastErrorInfo),0,SIZEOF(gMain.Services.Cert.Internal.LastErrorInfo));
	END_IF;

END_ACTION
```

#### Email.st - not listed in the package file held
```iecst
ACTION Email:

	gMain.Services.Email.In.Par.Port 															:= gPar.Services.Email.Port;
	gMain.Services.Email.In.Par.Timeout 														:= gPar.Services.Email.Timeout;
	gMain.Services.Email.In.Par.Host 															:= gPar.Services.Email.Host;
	gMain.Services.Email.In.Par.User 															:= gPar.Services.Email.User;
	gMain.Services.Email.In.Par.Password 														:= gPar.Services.Email.Password;
	gMain.Services.Email.In.Par.Sender 															:= gPar.Services.Email.Sender;
	gMain.Services.Email.In.Par.Receiver 														:= gPar.Services.Email.Receiver;
	gMain.Services.Email.In.Par.SSLConfigIdent													:= gMain.Services.Cert.SSLConfigIdent;

	gMain.Services.Email.In.Par.Subject															:= 'Automated Email Notification - Do Not Respond';
	gMain.Services.Email.In.Par.Text															:= 'Testing';

	IF gMain.Services.Email.In.Cmd.Reset THEN
		gMain.Services.Email.In.Cmd.Reset														:= FALSE;
		gMain.Services.Email.Internal.State														:= EMAIL_RESET_C;
	END_IF;

	brsmemset(ADR(gMain.Services.Email.Out),0,SIZEOF(gMain.Services.Email.Out));
	CASE gMain.Services.Email.Internal.State OF
		EMAIL_RESET_C:
			gMain.Services.Email.Out.Status.CurrentState										:= 'EMAIL_RESET_C';
			gMain.Services.Email.Out.Status.InReset												:= TRUE;
			brsmemset(ADR(gMain.Services.Email.In),0,SIZEOF(gMain.Services.Email.In));
			brsmemset(ADR(gMain.Services.Email.Internal),0,SIZEOF(gMain.Services.Email.Internal));
			gMain.Services.Email.Internal.State 												:= EMAIL_CHECKPARREADY_W;
		EMAIL_CHECKPARREADY_W:
			gMain.Services.Email.Out.Status.CurrentState										:= 'EMAIL_CHECKPARREADY_W';
			gMain.Services.Email.Out.Status.Initializing										:= TRUE;
			gMain.Services.Email.Internal.CTON_Timeout.IN 										:= TRUE;
			gMain.Services.Email.Internal.CTON_Timeout.PT 										:= LREAL_TO_TIME(30.0*1000.0); //Hardcoded because parameters are not yet loaded

			IF gMain.Services.Recipes.Out.ParametersReady THEN
				gMain.Services.Email.Internal.State 											:= EMAIL_IDLE_I;
			ELSIF gMain.Services.Email.Internal.CTON_Timeout.Q THEN
				gMain.Services.Email.Out.Status.Error 											:= TRUE;
				gMain.Services.Email.Out.ErrorInfo.Severity										:= 1;
				gMain.Services.Email.Out.ErrorInfo.Text 										:= 'Timeout';
				gMain.Services.Email.Out.ErrorInfo.State 										:= gMain.Services.Email.Out.Status.CurrentState;
				gMain.Services.Email.Internal.State 											:= EMAIL_ERROR_I;
			END_IF;
		EMAIL_IDLE_I:
			gMain.Services.Email.Out.Status.CurrentState										:= 'EMAIL_IDLE_I';
			gMain.Services.Email.Out.Status.WaitingForCommand									:= TRUE;

			IF gMain.Services.Email.In.Cmd.Send THEN
				gMain.Services.Email.In.Cmd.Send												:= FALSE;
				gMain.Services.Email.Internal.State 											:= EMAIL_SEND_D;
			END_IF;
		EMAIL_SEND_D:
			gMain.Services.Email.Out.Status.CurrentState										:= 'EMAIL_SEND_D';
			gMain.Services.Email.Out.Status.Processing											:= TRUE;
			gMain.Services.Email.Internal.CTON_Delay.IN 										:= TRUE;
			gMain.Services.Email.Internal.CTON_Delay.PT 										:= LREAL_TO_TIME(0.0*1000.0);

			IF gMain.Services.Email.Internal.CTON_Delay.Q OR 0.0 < 0.0001 THEN
				gMain.Services.Email.Internal.State 											:= EMAIL_SEND_C;
			END_IF;
		EMAIL_SEND_C:
			gMain.Services.Email.Out.Status.CurrentState										:= 'EMAIL_SEND_C';
			gMain.Services.Email.Out.Status.Processing											:= TRUE;
			gMain.Services.Email.Internal.SmtpsSend_0.enable									:= TRUE;
			gMain.Services.Email.Internal.SmtpsSend_0.port										:= gMain.Services.Email.In.Par.Port;
			gMain.Services.Email.Internal.SmtpsSend_0.timeout									:= gMain.Services.Email.In.Par.Timeout;
			gMain.Services.Email.Internal.SmtpsSend_0.pHost										:= ADR(gMain.Services.Email.In.Par.Host);
			gMain.Services.Email.Internal.SmtpsSend_0.pUser										:= ADR(gMain.Services.Email.In.Par.User);
			gMain.Services.Email.Internal.SmtpsSend_0.pPassword									:= ADR(gMain.Services.Email.In.Par.Password);
			gMain.Services.Email.Internal.SmtpsSend_0.pSender									:= ADR(gMain.Services.Email.In.Par.Sender);
			gMain.Services.Email.Internal.SmtpsSend_0.pReceiver									:= ADR(gMain.Services.Email.In.Par.Receiver);
			gMain.Services.Email.Internal.SmtpsSend_0.pSubject									:= ADR(gMain.Services.Email.In.Par.Subject);
			gMain.Services.Email.Internal.SmtpsSend_0.pText										:= ADR(gMain.Services.Email.In.Par.Text);
			gMain.Services.Email.Internal.SmtpsSend_0.attcnt									:= gMain.Services.Email.In.Par.AttachmentCount;
			gMain.Services.Email.Internal.SmtpsSend_0.pAttachment								:= gMain.Services.Email.In.Par.pAttachment;
			gMain.Services.Email.Internal.SmtpsSend_0.pDomain									:= ADR('gmail.com');
			gMain.Services.Email.Internal.SmtpsSend_0.sslCfgIdent								:= gMain.Services.Email.In.Par.SSLConfigIdent;
			gMain.Services.Email.Internal.State 												:= EMAIL_SEND_W;
		EMAIL_SEND_W:
			gMain.Services.Email.Out.Status.CurrentState										:= 'EMAIL_SEND_W';
			gMain.Services.Email.Out.Status.Processing											:= TRUE;
			gMain.Services.Email.Internal.CTON_Timeout.IN 										:= TRUE;
			gMain.Services.Email.Internal.CTON_Timeout.PT 										:= LREAL_TO_TIME(30.0*1000.0);

			IF gMain.Services.Email.Internal.SmtpsSend_0.status = 0 THEN
				gMain.Services.Email.Internal.SmtpsSend_0.enable								:= FALSE;
				gMain.Services.Email.Internal.State 											:= EMAIL_RESET_C;
			ELSIF gMain.Services.Email.Internal.SmtpsSend_0.status <> 65535 AND gMain.Services.Email.Internal.SmtpsSend_0.status <> 65534 THEN
				gMain.Services.Email.Internal.SmtpsSend_0.enable								:= FALSE;
				gMain.Services.Email.Out.Status.Error 											:= TRUE;
				gMain.Services.Email.Out.ErrorInfo.Severity										:= 2;
				gMain.Services.Email.Out.ErrorInfo.Code											:= gMain.Services.Email.Internal.SmtpsSend_0.status;
				gMain.Services.Email.Out.ErrorInfo.Text 										:= 'FBError';
				gMain.Services.Email.Out.ErrorInfo.State										:= gMain.Services.Email.Out.Status.CurrentState;
				gMain.Services.Email.Internal.State 											:= EMAIL_ERROR_I;
			ELSIF gMain.Services.Email.Internal.CTON_Timeout.Q THEN
				gMain.Services.Email.Internal.SmtpsSend_0.enable								:= FALSE;
				gMain.Services.Email.Out.Status.Error 											:= TRUE;
				gMain.Services.Email.Out.ErrorInfo.Severity										:= 2;
				gMain.Services.Email.Out.ErrorInfo.Text 										:= 'Timeout';
				gMain.Services.Email.Internal.State 											:= EMAIL_ERROR_I;
			END_IF;
		EMAIL_ERROR_I:
			gMain.Services.Email.Out.Status.CurrentState										:= 'EMAIL_ERROR_I';
			gMain.Services.Email.Out.Status.InError 											:= TRUE;
			IF gMain.ErrorReset THEN
				gMain.Services.Email.Internal.State 											:= EMAIL_RESET_C;
			END_IF;
	END_CASE;
	//Check for Commands that are still true. If they are still true then they were not handled and we need to error.
	IF NOT gMain.Services.Email.Out.Status.WaitingForCommand THEN
		IF gMain.Services.Email.In.Cmd.Send THEN
			gMain.Services.Email.In.Cmd.Send													:= FALSE;
			gMain.Services.Email.Out.IgnoreInfo.Cmd												:= 'Send';
			gMain.Services.Email.Out.IgnoreInfo.Reason											:= 'NotReady';
			gMain.Services.Email.Out.ErrorInfo.State											:= gMain.Services.Email.Out.Status.CurrentState;

			gMain.Services.Email.Internal.tempAlarm.name										:= 'EmailCmdIgnored';
			gMain.Services.Email.Internal.tempAlarm.allowMultiple								:= TRUE;
			gMain.Services.Email.Internal.tempAlarm.addText[0]									:= gMain.Services.Email.Out.IgnoreInfo.Cmd;
			gMain.Services.Email.Internal.tempAlarm.addText[1]									:= gMain.Services.Email.Out.IgnoreInfo.Reason;
			TC_Array_AddTop(ADR(gMain.Services.Alarms.In.AlarmList), SIZEOF(gMain.Services.Alarms.In.AlarmList), ADR(gMain.Services.Email.Internal.tempAlarm), SIZEOF(gMain.Services.Email.Internal.tempAlarm));
		END_IF;
	END_IF;
	brsmemset(ADR(gMain.Services.Email.Internal.BlankCmdCmp),0,SIZEOF(gMain.Services.Email.Internal.BlankCmdCmp));
	IF brsmemcmp(ADR(gMain.Services.Email.Internal.BlankCmdCmp),ADR(gMain.Services.Email.In.Cmd),SIZEOF(gMain.Services.Email.In.Cmd)) <> 0 THEN
		gMain.Services.Email.Out.ErrorInfo.State												:= gMain.Services.Email.Out.Status.CurrentState;

		gMain.Services.Email.Internal.tempAlarm.name											:= 'EmailUnhandledCmd';
		gMain.Services.Email.Internal.tempAlarm.allowMultiple									:= TRUE;
		gMain.Services.Email.Internal.tempAlarm.addText[0]										:= gMain.Services.Email.Out.ErrorInfo.State;
		TC_Array_AddTop(ADR(gMain.Services.Alarms.In.AlarmList), SIZEOF(gMain.Services.Alarms.In.AlarmList), ADR(gMain.Services.Email.Internal.tempAlarm), SIZEOF(gMain.Services.Email.Internal.tempAlarm));
	END_IF;
	brsmemset(ADR(gMain.Services.Email.In.Cmd),0,SIZEOF(gMain.Services.Email.In.Cmd));

	//Reset Timeout On State Change
	IF gMain.Services.Email.Internal.LastState <> gMain.Services.Email.Internal.State OR gMain.Services.Email.Internal.State = EMAIL_RESET_C THEN
		gMain.Services.Email.Internal.LastState													:= gMain.Services.Email.Internal.State;
		gMain.Services.Email.Internal.CTON_Timeout.IN											:= FALSE;
		gMain.Services.Email.Internal.CTON_Delay.IN												:= FALSE;
	END_IF;

	//Function Calls
	gMain.Services.Email.Internal.CTON_Timeout	(PAUSE := FALSE);
	gMain.Services.Email.Internal.CTON_Delay	(PAUSE := FALSE);
	gMain.Services.Email.Internal.SmtpsSend_0	();

	//Error Collection
	IF gMain.Services.Email.Out.Status.Error THEN
		IF brsmemcmp(ADR(gMain.Services.Email.Internal.LastErrorInfo),ADR(gMain.Services.Email.Out.ErrorInfo),SIZEOF(gMain.Services.Email.Internal.LastErrorInfo)) <> 0 THEN
			brsmemcpy(ADR(gMain.Services.Email.Internal.LastErrorInfo),ADR(gMain.Services.Email.Out.ErrorInfo),SIZEOF(gMain.Services.Email.Internal.LastErrorInfo));
			CASE gMain.Services.Email.Out.ErrorInfo.Severity OF
				1:
					gMain.Services.Email.Internal.tempAlarm.name				:= 'EmailSeverity1';
					gMain.Services.Email.Internal.tempAlarm.allowMultiple		:= TRUE;
					gMain.Services.Email.Internal.tempAlarm.addText[0]			:= gMain.Services.Email.Out.ErrorInfo.State;
					gMain.Services.Email.Internal.tempAlarm.addText[1]			:= gMain.Services.Email.Out.ErrorInfo.Text;

					TC_Array_AddTop(ADR(gMain.Services.Alarms.In.AlarmList), SIZEOF(gMain.Services.Alarms.In.AlarmList), ADR(gMain.Services.Email.Internal.tempAlarm), SIZEOF(gMain.Services.Email.Internal.tempAlarm));
				2:
					gMain.Services.Email.Internal.tempAlarm.name				:= 'EmailSeverity2';
					gMain.Services.Email.Internal.tempAlarm.allowMultiple		:= TRUE;
					gMain.Services.Email.Internal.tempAlarm.addText[0]			:= gMain.Services.Email.Out.ErrorInfo.State;
					gMain.Services.Email.Internal.tempAlarm.addText[1]			:= gMain.Services.Email.Out.ErrorInfo.Text;
					brsitoa(gMain.Services.Email.Out.ErrorInfo.Code, ADR(gMain.Services.Email.Internal.tempAlarm.addText[2]));

					TC_Array_AddTop(ADR(gMain.Services.Alarms.In.AlarmList), SIZEOF(gMain.Services.Alarms.In.AlarmList), ADR(gMain.Services.Email.Internal.tempAlarm), SIZEOF(gMain.Services.Email.Internal.tempAlarm));
				3:
					gMain.Services.Email.Internal.tempAlarm.name				:= 'EmailSeverity3';
					gMain.Services.Email.Internal.tempAlarm.allowMultiple		:= TRUE;
					gMain.Services.Email.Internal.tempAlarm.addText[0]			:= gMain.Services.Email.Out.ErrorInfo.State;
					gMain.Services.Email.Internal.tempAlarm.addText[1]			:= gMain.Services.Email.Out.ErrorInfo.Text;

					TC_Array_AddTop(ADR(gMain.Services.Alarms.In.AlarmList), SIZEOF(gMain.Services.Alarms.In.AlarmList), ADR(gMain.Services.Email.Internal.tempAlarm), SIZEOF(gMain.Services.Email.Internal.tempAlarm));
				4:
					gMain.Services.Email.Internal.tempAlarm.name				:= 'EmailSeverity4';
					gMain.Services.Email.Internal.tempAlarm.allowMultiple		:= TRUE;
					gMain.Services.Email.Internal.tempAlarm.addText[0]			:= gMain.Services.Email.Out.ErrorInfo.State;
					gMain.Services.Email.Internal.tempAlarm.addText[1]			:= gMain.Services.Email.Out.ErrorInfo.Text;

					TC_Array_AddTop(ADR(gMain.Services.Alarms.In.AlarmList), SIZEOF(gMain.Services.Alarms.In.AlarmList), ADR(gMain.Services.Email.Internal.tempAlarm), SIZEOF(gMain.Services.Email.Internal.tempAlarm));
			END_CASE;
		END_IF;
	ELSE
		brsmemset(ADR(gMain.Services.Email.Internal.LastErrorInfo),0,SIZEOF(gMain.Services.Email.Internal.LastErrorInfo));
	END_IF;

END_ACTION
```

### Program Logical/Vis (IEC)

#### Main.st - Init, cyclic, exit code
```iecst
PROGRAM _INIT

END_PROGRAM

PROGRAM _CYCLIC

	Vis_General;
	Header;
	Footer;
	Navigation;
	Services_DirMan;
	Settings;
	Alarms_Active;
	Alarms_History;

END_PROGRAM

PROGRAM _EXIT

END_PROGRAM
```

#### Variables.var - Local variables
```iecst
VAR
	Idx_FileList : INT;
	Idx_AlarmList : INT;
END_VAR
```

#### Vis_General.st
```iecst
ACTION Vis_General:

END_ACTION
```

#### Header.st
```iecst
ACTION Header:

//Monitor
	gVis.Header.Monitor.Styles.Text											:= '#888888';
	gVis.Header.Monitor.Styles.Background									:= '#111111';
	gVis.Header.Monitor.Styles.GridColor									:= '#888888';
	gVis.Header.Monitor.Styles.Line0										:= '#00FF00';
	gVis.Header.Monitor.Styles.Line1										:= '#FFFF00';
	gVis.Header.Monitor.Styles.Line2										:= '#FF00FF';
	gVis.Header.Monitor.Styles.Line3										:= '#00FFFF';

//Notifications
	gVis.Header.Notifications.Visible[0]									:= gMain.Services.Alarms.Out.AlarmActive;
	gVis.Header.Notifications.Visible[1]									:= gMain.Services.Alarms.Out.AlarmActive;
	gVis.Header.Notifications.Visible[2]									:= gVis.Settings.Save.Modified;
	gVis.Header.Notifications.Visible[3]									:= gIO.ForceEnable;

END_ACTION
```

#### Footer.st
```iecst
ACTION Footer:

	gVis.Footer.IdentifyConfig_0();
	gVis.Footer.Revision 													:= gVis.Footer.IdentifyConfig_0.ConfigID;
	brsstrcat(ADR(gVis.Footer.Revision),ADR(' - '));
	brsstrcat(ADR(gVis.Footer.Revision),ADR(gVis.Footer.IdentifyConfig_0.ConfigVersion));

	gVis.Footer.currentTime													:= gMain.Services.Time.Out.Status.CurrentTime;

	IF gVis.Footer.CTON_Init.Q AND gMain.Services.Time.Out.Status.TimeValid = FALSE THEN
		gVis.Footer.TimeNotValid := TRUE;
	ELSE
		gVis.Footer.TimeNotValid := FALSE;
	END_IF

	//Handle Time
	IF gVis.Footer.SetTime THEN
		gVis.Footer.SetTime 												:= FALSE;
		gMain.Services.Time.In.Cmd.setTime									:= TRUE;
		gMain.Services.Time.In.Par.newTime									:= gVis.Footer.newTime;
	END_IF

	IF gVis.Footer.Start THEN
		gMain.Process.Master.In.Cmd.Start									:= TRUE;
	END_IF;
	gVis.Footer.Start														:= FALSE;
	IF gVis.Footer.Pause THEN
		gMain.Process.Master.In.Cmd.Pause									:= TRUE;
	END_IF;
	gVis.Footer.Pause														:= FALSE;
	IF gVis.Footer.Stop THEN
		gMain.Process.Master.In.Cmd.NormalStop								:= TRUE;
	END_IF;
	gVis.Footer.Stop														:= FALSE;

	gVis.Footer.CTON_Init(IN:=TRUE, PT:=T#5s);

END_ACTION
```

#### Navigation.st
```iecst
ACTION Navigation:
	IF gVis.Navigation.STOP THEN
		gVis.Navigation.STOP := FALSE;
		gIO.Safety.TC_IO_DI_HMI_STOP.IOMapping 		:= TRUE;
		gIO.Safety.TC_IO_DI_HMI_STOP.Sim.Logical 	:= TRUE;
	ELSIF gMain.ErrorReset THEN
		gIO.Safety.TC_IO_DI_HMI_STOP.IOMapping 		:= FALSE;
		gIO.Safety.TC_IO_DI_HMI_STOP.Sim.Logical 	:= FALSE;
	END_IF;
END_ACTION
```
